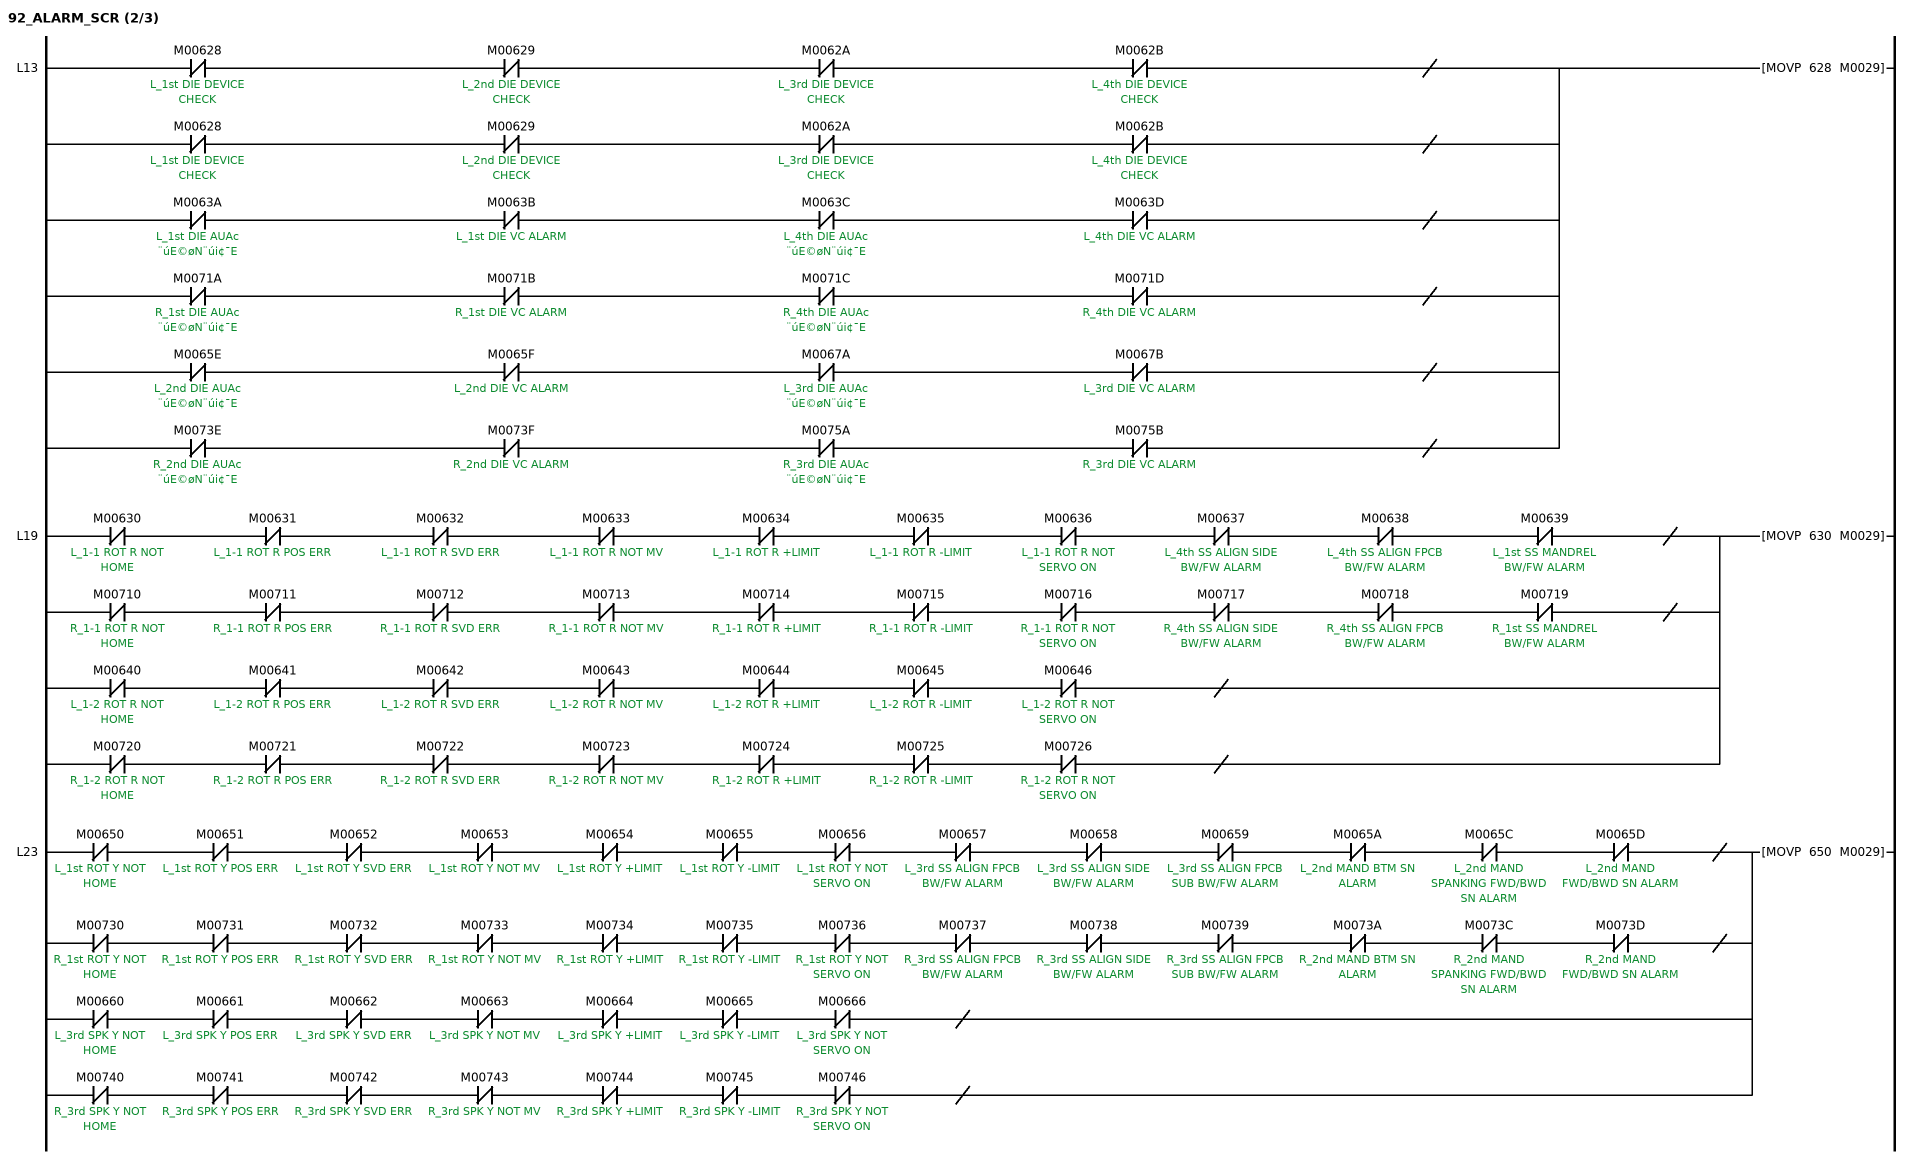
[picture p432: 92_ALARM_SCR rungs L13-L23]
; L13
LOAD NOT  M00628	// L_1st DIE DEVICE CHECK
AND NOT   M00629	// L_2nd DIE DEVICE CHECK
AND NOT   M0062A	// L_3rd DIE DEVICE CHECK
AND NOT   M0062B	// L_4th DIE DEVICE CHECK
NOT
LOAD NOT  M00628	// L_1st DIE DEVICE CHECK
AND NOT   M00629	// L_2nd DIE DEVICE CHECK
AND NOT   M0062A	// L_3rd DIE DEVICE CHECK
AND NOT   M0062B	// L_4th DIE DEVICE CHECK
NOT
OR LOAD
LOAD NOT  M0063A	// L_1st DIE AUAc ¨úE©øN¨úi¢¯E
AND NOT   M0063B	// L_1st DIE VC ALARM
AND NOT   M0063C	// L_4th DIE AUAc ¨úE©øN¨úi¢¯E
AND NOT   M0063D	// L_4th DIE VC ALARM
NOT
OR LOAD
LOAD NOT  M0071A	// R_1st DIE AUAc ¨úE©øN¨úi¢¯E
AND NOT   M0071B	// R_1st DIE VC ALARM
AND NOT   M0071C	// R_4th DIE AUAc ¨úE©øN¨úi¢¯E
AND NOT   M0071D	// R_4th DIE VC ALARM
NOT
OR LOAD
LOAD NOT  M0065E	// L_2nd DIE AUAc ¨úE©øN¨úi¢¯E
AND NOT   M0065F	// L_2nd DIE VC ALARM
AND NOT   M0067A	// L_3rd DIE AUAc ¨úE©øN¨úi¢¯E
AND NOT   M0067B	// L_3rd DIE VC ALARM
NOT
OR LOAD
LOAD NOT  M0073E	// R_2nd DIE AUAc ¨úE©øN¨úi¢¯E
AND NOT   M0073F	// R_2nd DIE VC ALARM
AND NOT   M0075A	// R_3rd DIE AUAc ¨úE©øN¨úi¢¯E
AND NOT   M0075B	// R_3rd DIE VC ALARM
NOT
OR LOAD
MOVP      628 M0029
; L19
LOAD NOT  M00630	// L_1-1 ROT R NOT HOME
AND NOT   M00631	// L_1-1 ROT R POS ERR
AND NOT   M00632	// L_1-1 ROT R SVD ERR
AND NOT   M00633	// L_1-1 ROT R NOT MV
AND NOT   M00634	// L_1-1 ROT R +LIMIT
AND NOT   M00635	// L_1-1 ROT R -LIMIT
AND NOT   M00636	// L_1-1 ROT R NOT SERVO ON
AND NOT   M00637	// L_4th SS ALIGN SIDE BW/FW ALARM
AND NOT   M00638	// L_4th SS ALIGN FPCB BW/FW ALARM
AND NOT   M00639	// L_1st SS MANDREL BW/FW ALARM
NOT
LOAD NOT  M00710	// R_1-1 ROT R NOT HOME
AND NOT   M00711	// R_1-1 ROT R POS ERR
AND NOT   M00712	// R_1-1 ROT R SVD ERR
AND NOT   M00713	// R_1-1 ROT R NOT MV
AND NOT   M00714	// R_1-1 ROT R +LIMIT
AND NOT   M00715	// R_1-1 ROT R -LIMIT
AND NOT   M00716	// R_1-1 ROT R NOT SERVO ON
AND NOT   M00717	// R_4th SS ALIGN SIDE BW/FW ALARM
AND NOT   M00718	// R_4th SS ALIGN FPCB BW/FW ALARM
AND NOT   M00719	// R_1st SS MANDREL BW/FW ALARM
NOT
OR LOAD
LOAD NOT  M00640	// L_1-2 ROT R NOT HOME
AND NOT   M00641	// L_1-2 ROT R POS ERR
AND NOT   M00642	// L_1-2 ROT R SVD ERR
AND NOT   M00643	// L_1-2 ROT R NOT MV
AND NOT   M00644	// L_1-2 ROT R +LIMIT
AND NOT   M00645	// L_1-2 ROT R -LIMIT
AND NOT   M00646	// L_1-2 ROT R NOT SERVO ON
NOT
OR LOAD
LOAD NOT  M00720	// R_1-2 ROT R NOT HOME
AND NOT   M00721	// R_1-2 ROT R POS ERR
AND NOT   M00722	// R_1-2 ROT R SVD ERR
AND NOT   M00723	// R_1-2 ROT R NOT MV
AND NOT   M00724	// R_1-2 ROT R +LIMIT
AND NOT   M00725	// R_1-2 ROT R -LIMIT
AND NOT   M00726	// R_1-2 ROT R NOT SERVO ON
NOT
OR LOAD
MOVP      630 M0029
; L23
LOAD NOT  M00650	// L_1st ROT Y NOT HOME
AND NOT   M00651	// L_1st ROT Y POS ERR
AND NOT   M00652	// L_1st ROT Y SVD ERR
AND NOT   M00653	// L_1st ROT Y NOT MV
AND NOT   M00654	// L_1st ROT Y +LIMIT
AND NOT   M00655	// L_1st ROT Y -LIMIT
AND NOT   M00656	// L_1st ROT Y NOT SERVO ON
AND NOT   M00657	// L_3rd SS ALIGN FPCB BW/FW ALARM
AND NOT   M00658	// L_3rd SS ALIGN SIDE BW/FW ALARM
AND NOT   M00659	// L_3rd SS ALIGN FPCB SUB BW/FW ALARM
AND NOT   M0065A	// L_2nd MAND BTM SN ALARM
AND NOT   M0065C	// L_2nd MAND SPANKING FWD/BWD SN ALARM
AND NOT   M0065D	// L_2nd MAND FWD/BWD SN ALARM
NOT
LOAD NOT  M00730	// R_1st ROT Y NOT HOME
AND NOT   M00731	// R_1st ROT Y POS ERR
AND NOT   M00732	// R_1st ROT Y SVD ERR
AND NOT   M00733	// R_1st ROT Y NOT MV
AND NOT   M00734	// R_1st ROT Y +LIMIT
AND NOT   M00735	// R_1st ROT Y -LIMIT
AND NOT   M00736	// R_1st ROT Y NOT SERVO ON
AND NOT   M00737	// R_3rd SS ALIGN FPCB BW/FW ALARM
AND NOT   M00738	// R_3rd SS ALIGN SIDE BW/FW ALARM
AND NOT   M00739	// R_3rd SS ALIGN FPCB SUB BW/FW ALARM
AND NOT   M0073A	// R_2nd MAND BTM SN ALARM
AND NOT   M0073C	// R_2nd MAND SPANKING FWD/BWD SN ALARM
AND NOT   M0073D	// R_2nd MAND FWD/BWD SN ALARM
NOT
OR LOAD
LOAD NOT  M00660	// L_3rd SPK Y NOT HOME
AND NOT   M00661	// L_3rd SPK Y POS ERR
AND NOT   M00662	// L_3rd SPK Y SVD ERR
AND NOT   M00663	// L_3rd SPK Y NOT MV
AND NOT   M00664	// L_3rd SPK Y +LIMIT
AND NOT   M00665	// L_3rd SPK Y -LIMIT
AND NOT   M00666	// L_3rd SPK Y NOT SERVO ON
NOT
OR LOAD
LOAD NOT  M00740	// R_3rd SPK Y NOT HOME
AND NOT   M00741	// R_3rd SPK Y POS ERR
AND NOT   M00742	// R_3rd SPK Y SVD ERR
AND NOT   M00743	// R_3rd SPK Y NOT MV
AND NOT   M00744	// R_3rd SPK Y +LIMIT
AND NOT   M00745	// R_3rd SPK Y -LIMIT
AND NOT   M00746	// R_3rd SPK Y NOT SERVO ON
NOT
OR LOAD
MOVP      650 M0029

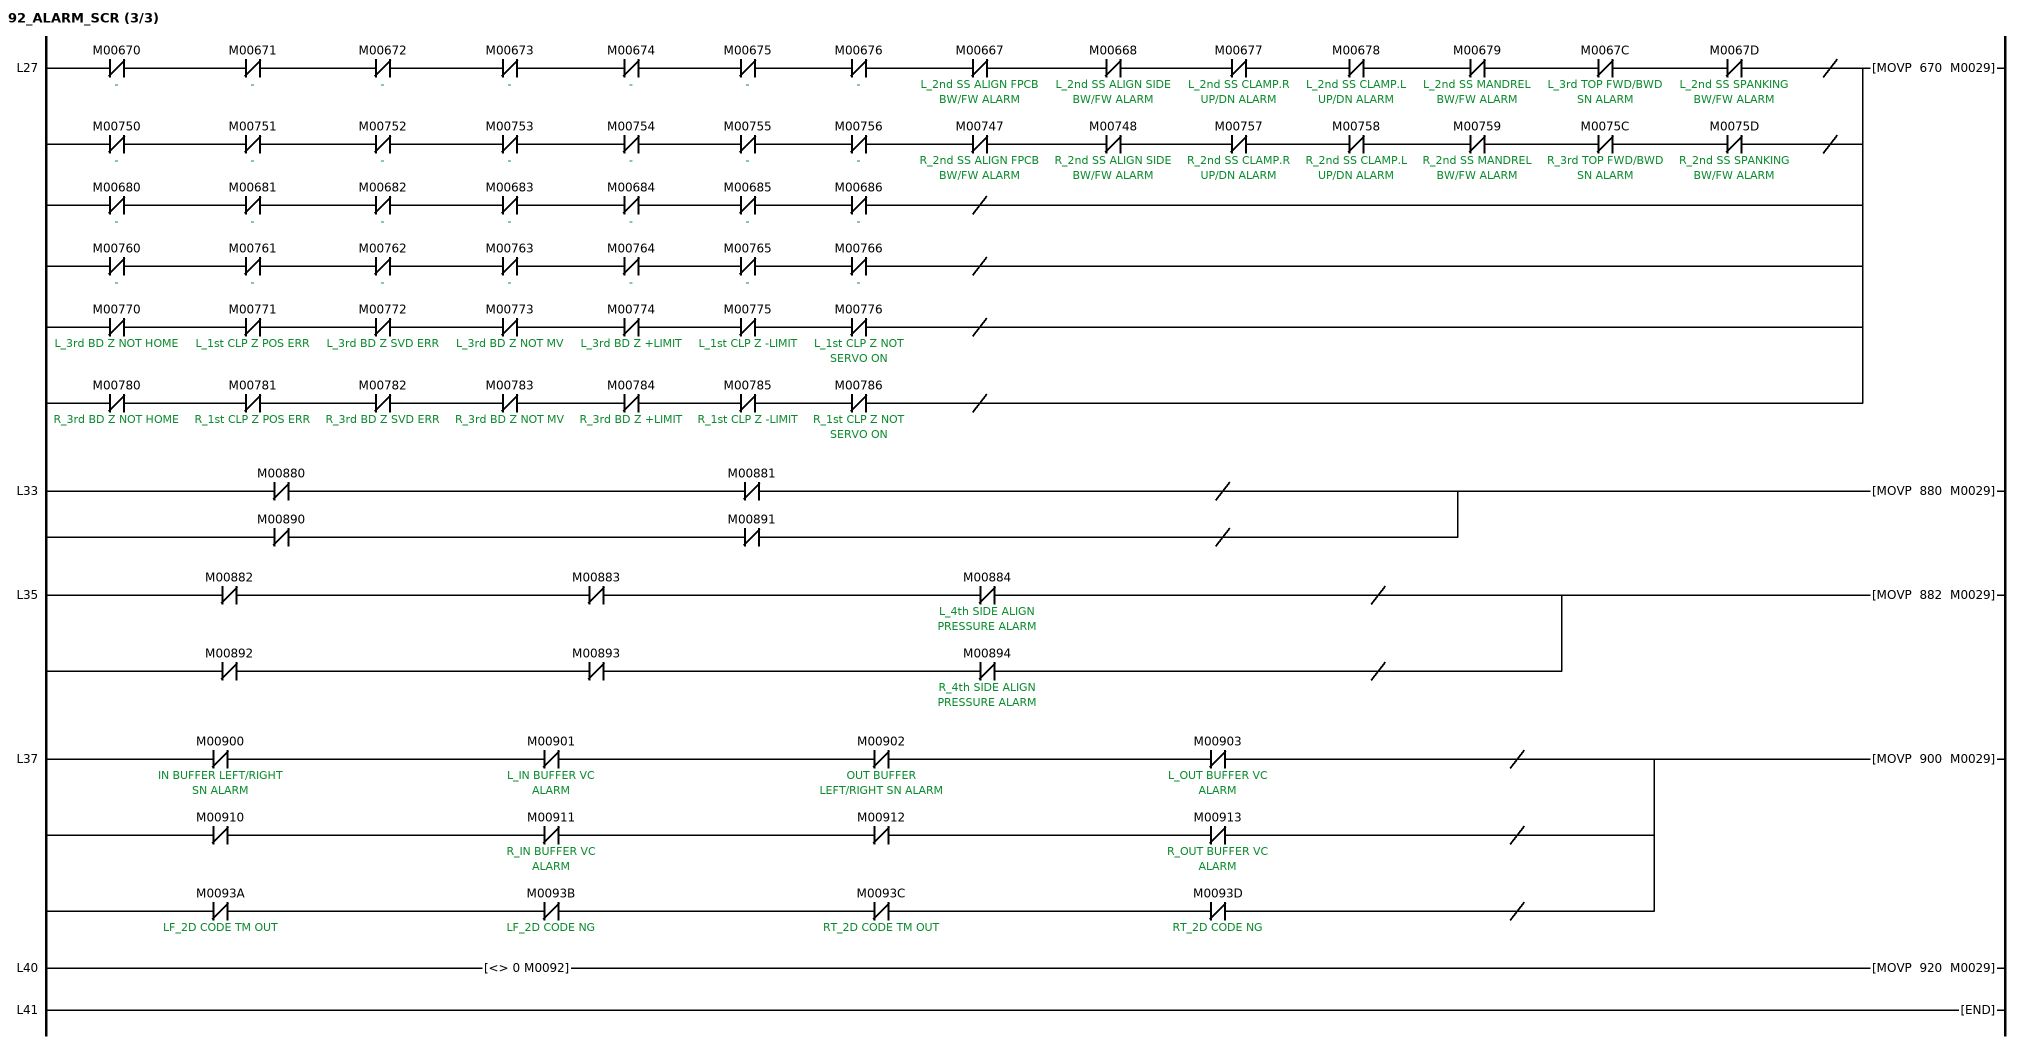
; L27
LOAD NOT  M00670	// -
AND NOT   M00671	// -
AND NOT   M00672	// -
AND NOT   M00673	// -
AND NOT   M00674	// -
AND NOT   M00675	// -
AND NOT   M00676	// -
AND NOT   M00667	// L_2nd SS ALIGN FPCB BW/FW ALARM
AND NOT   M00668	// L_2nd SS ALIGN SIDE BW/FW ALARM
AND NOT   M00677	// L_2nd SS CLAMP.R UP/DN ALARM
AND NOT   M00678	// L_2nd SS CLAMP.L UP/DN ALARM
AND NOT   M00679	// L_2nd SS MANDREL BW/FW ALARM
AND NOT   M0067C	// L_3rd TOP FWD/BWD SN ALARM
AND NOT   M0067D	// L_2nd SS SPANKING BW/FW ALARM
NOT
LOAD NOT  M00750	// -
AND NOT   M00751	// -
AND NOT   M00752	// -
AND NOT   M00753	// -
AND NOT   M00754	// -
AND NOT   M00755	// -
AND NOT   M00756	// -
AND NOT   M00747	// R_2nd SS ALIGN FPCB BW/FW ALARM
AND NOT   M00748	// R_2nd SS ALIGN SIDE BW/FW ALARM
AND NOT   M00757	// R_2nd SS CLAMP.R UP/DN ALARM
AND NOT   M00758	// R_2nd SS CLAMP.L UP/DN ALARM
AND NOT   M00759	// R_2nd SS MANDREL BW/FW ALARM
AND NOT   M0075C	// R_3rd TOP FWD/BWD SN ALARM
AND NOT   M0075D	// R_2nd SS SPANKING BW/FW ALARM
NOT
OR LOAD
LOAD NOT  M00680	// -
AND NOT   M00681	// -
AND NOT   M00682	// -
AND NOT   M00683	// -
AND NOT   M00684	// -
AND NOT   M00685	// -
AND NOT   M00686	// -
NOT
OR LOAD
LOAD NOT  M00760	// -
AND NOT   M00761	// -
AND NOT   M00762	// -
AND NOT   M00763	// -
AND NOT   M00764	// -
AND NOT   M00765	// -
AND NOT   M00766	// -
NOT
OR LOAD
LOAD NOT  M00770	// L_3rd BD Z NOT HOME
AND NOT   M00771	// L_1st CLP Z POS ERR
AND NOT   M00772	// L_3rd BD Z SVD ERR
AND NOT   M00773	// L_3rd BD Z NOT MV
AND NOT   M00774	// L_3rd BD Z +LIMIT
AND NOT   M00775	// L_1st CLP Z -LIMIT
AND NOT   M00776	// L_1st CLP Z NOT SERVO ON
NOT
OR LOAD
LOAD NOT  M00780	// R_3rd BD Z NOT HOME
AND NOT   M00781	// R_1st CLP Z POS ERR
AND NOT   M00782	// R_3rd BD Z SVD ERR
AND NOT   M00783	// R_3rd BD Z NOT MV
AND NOT   M00784	// R_3rd BD Z +LIMIT
AND NOT   M00785	// R_1st CLP Z -LIMIT
AND NOT   M00786	// R_1st CLP Z NOT SERVO ON
NOT
OR LOAD
MOVP      670 M0029
; L33
LOAD NOT  M00880
AND NOT   M00881
NOT
LOAD NOT  M00890
AND NOT   M00891
NOT
OR LOAD
MOVP      880 M0029
; L35
LOAD NOT  M00882
AND NOT   M00883
AND NOT   M00884	// L_4th SIDE ALIGN PRESSURE ALARM
NOT
LOAD NOT  M00892
AND NOT   M00893
AND NOT   M00894	// R_4th SIDE ALIGN PRESSURE ALARM
NOT
OR LOAD
MOVP      882 M0029
; L37
LOAD NOT  M00900	// IN BUFFER LEFT/RIGHT SN ALARM
AND NOT   M00901	// L_IN BUFFER VC ALARM
AND NOT   M00902	// OUT BUFFER LEFT/RIGHT SN ALARM
AND NOT   M00903	// L_OUT BUFFER VC ALARM
NOT
LOAD NOT  M00910
AND NOT   M00911	// R_IN BUFFER VC ALARM
AND NOT   M00912
AND NOT   M00913	// R_OUT BUFFER VC ALARM
NOT
OR LOAD
LOAD NOT  M0093A	// LF_2D CODE TM OUT
AND NOT   M0093B	// LF_2D CODE NG
AND NOT   M0093C	// RT_2D CODE TM OUT
AND NOT   M0093D	// RT_2D CODE NG
NOT
OR LOAD
MOVP      900 M0029
; L40
LOAD<>    0 M0092
MOVP      920 M0029
; L41
END

PROGRAM AUTO_LOAD (task: ¨ö¨¬A¥ì CA¡¤I¡¾¡¿¡¤¡Í)

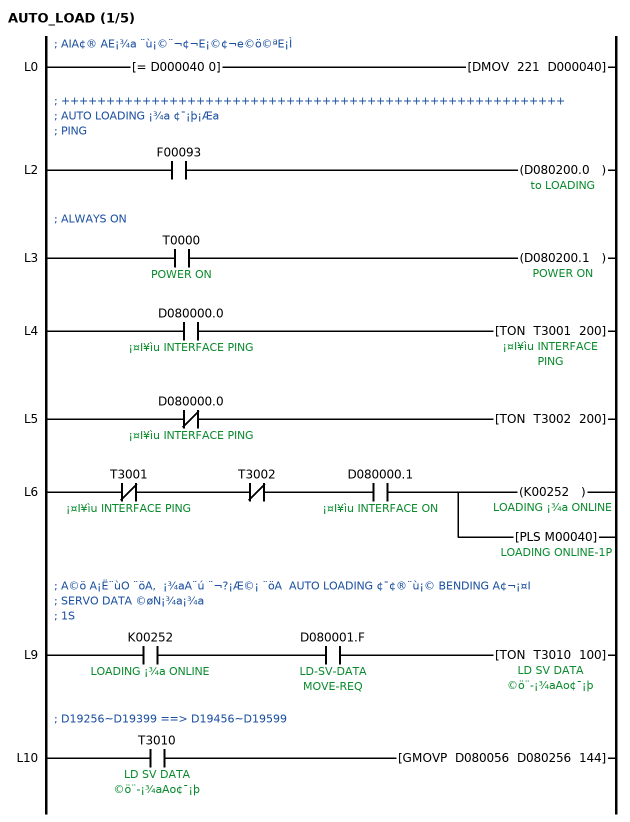
; L0
LOAD=     D000040 0
DMOV      221 D000040
// output comment: AIA¢® AE¡¾a ¨ù¡©¨¬¢¬E¡©¢¬e©ö©ªE¡Ì
// ++++++++++++++++++++++++++++++++++++++++++++++++++++++++
//    AUTO LOADING ¡¾a ¢¯¡þ¡Æa
; L2
LOAD      F00093
OUT       D080200.0	// to LOADING
// output comment: PING
; L3
LOAD      T0000	// POWER ON
OUT       D080200.1	// POWER ON
// output comment: ALWAYS ON
; L4
LOAD      D080000.0	// ¡¤I¥ìu INTERFACE PING
TON       T3001 200	// ¡¤I¥ìu INTERFACE PING
; L5
LOAD NOT  D080000.0	// ¡¤I¥ìu INTERFACE PING
TON       T3002 200
; L6
LOAD NOT  T3001	// ¡¤I¥ìu INTERFACE PING
AND NOT   T3002
AND       D080000.1	// ¡¤I¥ìu INTERFACE ON
OUT       K00252	// LOADING ¡¾a ONLINE
OUTP      M00040	// LOADING ONLINE-1P
// A©ö A¡Ë¨ùO ¨öA,  ¡¾aA¨ú ¨¬?¡Æ©¡ ¨öA  AUTO LOADING ¢¯¢®¨ù¡© BENDING A¢¬¡¤I  SERVO DATA ©øN¡¾a¡¾a
; L9
LOAD      K00252	// LOADING ¡¾a ONLINE
AND       D080001.F	// LD-SV-DATA MOVE-REQ
TON       T3010 100	// LD SV DATA ©ö¨­¡¾aAo¢¯¡þ
// output comment: 1S
; L10
LOAD      T3010	// LD SV DATA ©ö¨­¡¾aAo¢¯¡þ
GMOVP     D080056 D080256 144
// output comment: D19256~D19399 ==> D19456~D19599

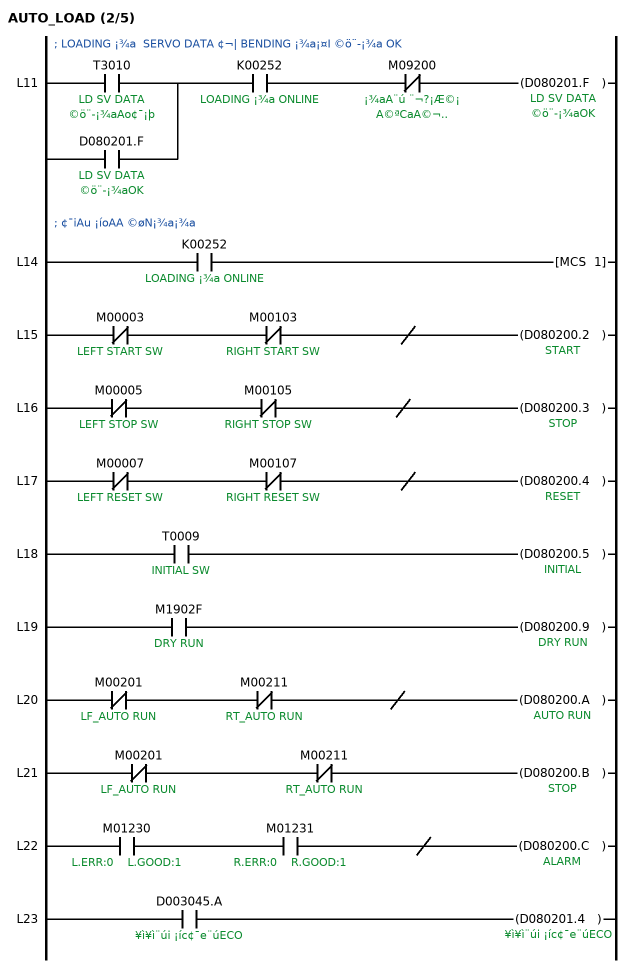
; L11
LOAD      T3010	// LD SV DATA ©ö¨­¡¾aAo¢¯¡þ
OR        D080201.F	// LD SV DATA ©ö¨­¡¾aOK
AND       K00252	// LOADING ¡¾a ONLINE
AND NOT   M09200	// ¡¾aA¨ú ¨¬?¡Æ©¡ A©ªCaA©¬..
OUT       D080201.F	// LD SV DATA ©ö¨­¡¾aOK
// output comment: LOADING ¡¾a  SERVO DATA ¢¬| BENDING ¡¾a¡¤I ©ö¨­¡¾a OK
// ¢¯iAu ¡íoAA ©øN¡¾a¡¾a
; L14
LOAD      K00252	// LOADING ¡¾a ONLINE
MCS       1
; L15
LOAD NOT  M00003	// LEFT START SW
AND NOT   M00103	// RIGHT START SW
NOT
OUT       D080200.2	// START
; L16
LOAD NOT  M00005	// LEFT STOP SW
AND NOT   M00105	// RIGHT STOP SW
NOT
OUT       D080200.3	// STOP
; L17
LOAD NOT  M00007	// LEFT RESET SW
AND NOT   M00107	// RIGHT RESET SW
NOT
OUT       D080200.4	// RESET
; L18
LOAD      T0009	// INITIAL SW
OUT       D080200.5	// INITIAL
; L19
LOAD      M1902F	// DRY RUN
OUT       D080200.9	// DRY RUN
; L20
LOAD NOT  M00201	// LF_AUTO RUN
AND NOT   M00211	// RT_AUTO RUN
NOT
OUT       D080200.A	// AUTO RUN
; L21
LOAD NOT  M00201	// LF_AUTO RUN
AND NOT   M00211	// RT_AUTO RUN
OUT       D080200.B	// STOP
; L22
LOAD      M01230	// L.ERR:0    L.GOOD:1
AND       M01231	// R.ERR:0    R.GOOD:1
NOT
OUT       D080200.C	// ALARM
; L23
LOAD      D003045.A	// ¥ì¥ì¨úi ¡íc¢¯e¨úECO
OUT       D080201.4	// ¥ì¥ì¨úi ¡íc¢¯e¨úECO

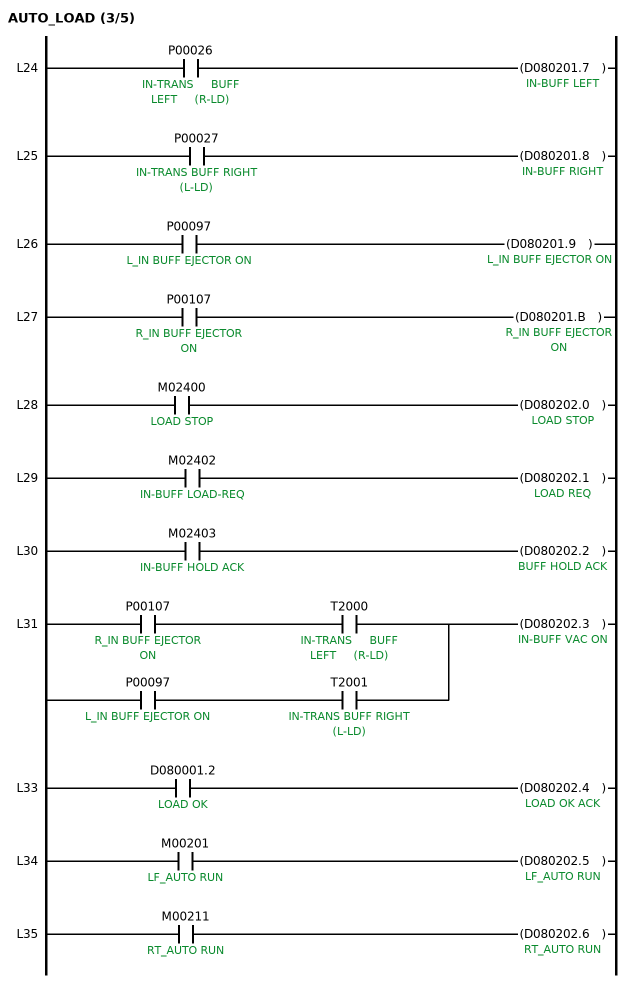
; L24
LOAD      P00026	// IN-TRANS     BUFF     LEFT     (R-LD)
OUT       D080201.7	// IN-BUFF LEFT
; L25
LOAD      P00027	// IN-TRANS BUFF RIGHT     (L-LD)
OUT       D080201.8	// IN-BUFF RIGHT
; L26
LOAD      P00097	// L_IN BUFF EJECTOR ON
OUT       D080201.9	// L_IN BUFF EJECTOR ON
; L27
LOAD      P00107	// R_IN BUFF EJECTOR ON
OUT       D080201.B	// R_IN BUFF EJECTOR ON
; L28
LOAD      M02400	// LOAD STOP
OUT       D080202.0	// LOAD STOP
; L29
LOAD      M02402	// IN-BUFF LOAD-REQ
OUT       D080202.1	// LOAD REQ
; L30
LOAD      M02403	// IN-BUFF HOLD ACK
OUT       D080202.2	// BUFF HOLD ACK
; L31
LOAD      P00107	// R_IN BUFF EJECTOR ON
AND       T2000	// IN-TRANS     BUFF     LEFT     (R-LD)
LOAD      P00097	// L_IN BUFF EJECTOR ON
AND       T2001	// IN-TRANS BUFF RIGHT     (L-LD)
OR LOAD
OUT       D080202.3	// IN-BUFF VAC ON
; L33
LOAD      D080001.2	// LOAD OK
OUT       D080202.4	// LOAD OK ACK
; L34
LOAD      M00201	// LF_AUTO RUN
OUT       D080202.5	// LF_AUTO RUN
; L35
LOAD      M00211	// RT_AUTO RUN
OUT       D080202.6	// RT_AUTO RUN

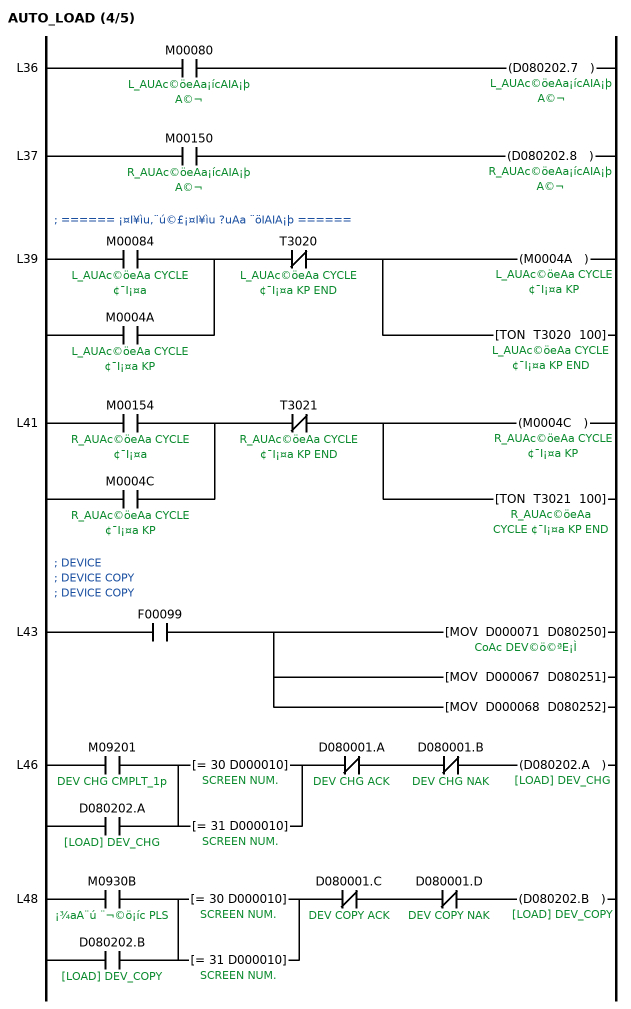
; L36
LOAD      M00080	// L_AUAc©öeAa¡ícAIA¡þA©¬
OUT       D080202.7	// L_AUAc©öeAa¡ícAIA¡þA©¬
; L37
LOAD      M00150	// R_AUAc©öeAa¡ícAIA¡þA©¬
OUT       D080202.8	// R_AUAc©öeAa¡ícAIA¡þA©¬
// ====== ¡¤I¥ìu,¨ú©£¡¤I¥ìu ?uAa ¨öIAIA¡þ ======
; L39
LOAD      M00084	// L_AUAc©öeAa CYCLE ¢¯I¡¤a
OR        M0004A	// L_AUAc©öeAa CYCLE ¢¯I¡¤a KP
AND NOT   T3020	// L_AUAc©öeAa CYCLE ¢¯I¡¤a KP END
OUT       M0004A	// L_AUAc©öeAa CYCLE ¢¯I¡¤a KP
TON       T3020 100	// L_AUAc©öeAa CYCLE ¢¯I¡¤a KP END
; L41
LOAD      M00154	// R_AUAc©öeAa CYCLE ¢¯I¡¤a
OR        M0004C	// R_AUAc©öeAa CYCLE ¢¯I¡¤a KP
AND NOT   T3021	// R_AUAc©öeAa CYCLE ¢¯I¡¤a KP END
OUT       M0004C	// R_AUAc©öeAa CYCLE ¢¯I¡¤a KP
TON       T3021 100	// R_AUAc©öeAa CYCLE ¢¯I¡¤a KP END
; L43
LOAD      F00099
MOV       D000071 D080250	// CoAc DEV©ö©ªE¡Ì
MOV       D000067 D080251
MOV       D000068 D080252
// output comment: DEVICE
// output comment: DEVICE COPY
// output comment: DEVICE COPY
; L46
LOAD      M09201	// DEV CHG CMPLT_1p
OR        D080202.A	// [LOAD] DEV_CHG
LOAD=     30 D000010	// SCREEN NUM.
OR=       31 D000010	// SCREEN NUM.
AND LOAD
AND NOT   D080001.A	// DEV CHG ACK
AND NOT   D080001.B	// DEV CHG NAK
OUT       D080202.A	// [LOAD] DEV_CHG
; L48
LOAD      M0930B	// ¡¾aA¨ú ¨¬©ö¡íc PLS
OR        D080202.B	// [LOAD] DEV_COPY
LOAD=     30 D000010	// SCREEN NUM.
OR=       31 D000010	// SCREEN NUM.
AND LOAD
AND NOT   D080001.C	// DEV COPY ACK
AND NOT   D080001.D	// DEV COPY NAK
OUT       D080202.B	// [LOAD] DEV_COPY

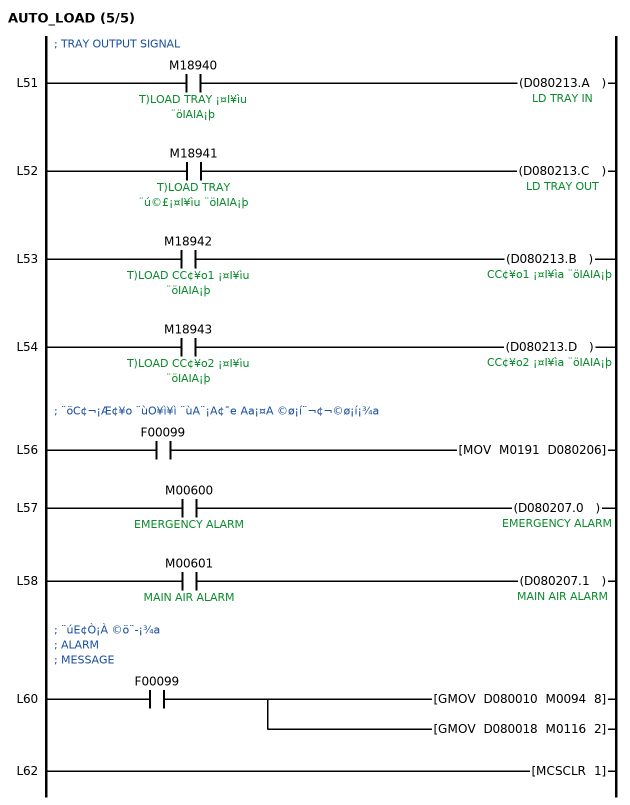
// TRAY OUTPUT SIGNAL
; L51
LOAD      M18940	// T)LOAD TRAY ¡¤I¥ìu ¨öIAIA¡þ
OUT       D080213.A	// LD TRAY IN
; L52
LOAD      M18941	// T)LOAD TRAY ¨ú©£¡¤I¥ìu ¨öIAIA¡þ
OUT       D080213.C	// LD TRAY OUT
; L53
LOAD      M18942	// T)LOAD CC¢¥o1 ¡¤I¥ìu ¨öIAIA¡þ
OUT       D080213.B	// CC¢¥o1 ¡¤I¥ìa ¨öIAIA¡þ
; L54
LOAD      M18943	// T)LOAD CC¢¥o2 ¡¤I¥ìu ¨öIAIA¡þ
OUT       D080213.D	// CC¢¥o2 ¡¤I¥ìa ¨öIAIA¡þ
// ¨öC¢¬¡Æ¢¥o ¨ùO¥ì¥ì ¨ùA¨¡A¢¯e Aa¡¤A ©ø¡í¨¬¢¬©ø¡í¡¾a
; L56
LOAD      F00099
MOV       M0191 D080206
; L57
LOAD      M00600	// EMERGENCY ALARM
OUT       D080207.0	// EMERGENCY ALARM
; L58
LOAD      M00601	// MAIN AIR ALARM
OUT       D080207.1	// MAIN AIR ALARM
// ¨úE¢Ò¡À ©ö¨­¡¾a
; L60
LOAD      F00099
GMOV      D080010 M0094 8
GMOV      D080018 M0116 2
// output comment: ALARM
// output comment: MESSAGE
; L62
MCSCLR    1

PROGRAM AUTO_UNLOAD (task: ¨ö¨¬A¥ì CA¡¤I¡¾¡¿¡¤¡Í)

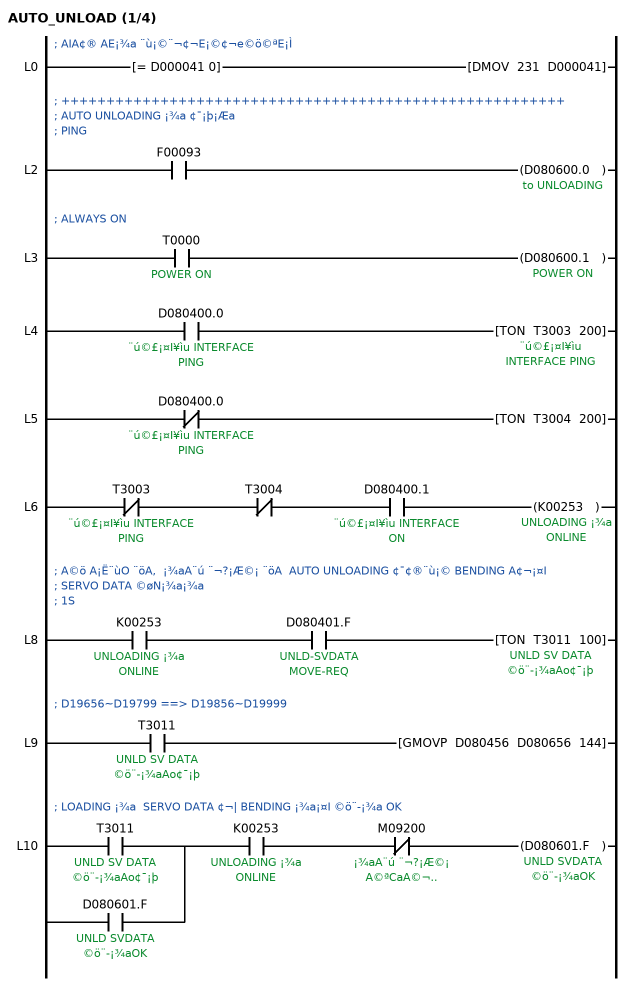
; L0
LOAD=     D000041 0
DMOV      231 D000041
// output comment: AIA¢® AE¡¾a ¨ù¡©¨¬¢¬E¡©¢¬e©ö©ªE¡Ì
// ++++++++++++++++++++++++++++++++++++++++++++++++++++++++
//    AUTO UNLOADING ¡¾a ¢¯¡þ¡Æa
; L2
LOAD      F00093
OUT       D080600.0	// to UNLOADING
// output comment: PING
; L3
LOAD      T0000	// POWER ON
OUT       D080600.1	// POWER ON
// output comment: ALWAYS ON
; L4
LOAD      D080400.0	// ¨ú©£¡¤I¥ìu INTERFACE PING
TON       T3003 200	// ¨ú©£¡¤I¥ìu INTERFACE PING
; L5
LOAD NOT  D080400.0	// ¨ú©£¡¤I¥ìu INTERFACE PING
TON       T3004 200
; L6
LOAD NOT  T3003	// ¨ú©£¡¤I¥ìu INTERFACE PING
AND NOT   T3004
AND       D080400.1	// ¨ú©£¡¤I¥ìu INTERFACE ON
OUT       K00253	// UNLOADING ¡¾a ONLINE
// A©ö A¡Ë¨ùO ¨öA,  ¡¾aA¨ú ¨¬?¡Æ©¡ ¨öA  AUTO UNLOADING ¢¯¢®¨ù¡© BENDING A¢¬¡¤I  SERVO DATA ©øN¡¾a¡¾a
; L8
LOAD      K00253	// UNLOADING ¡¾a ONLINE
AND       D080401.F	// UNLD-SVDATA MOVE-REQ
TON       T3011 100	// UNLD SV DATA ©ö¨­¡¾aAo¢¯¡þ
// output comment: 1S
; L9
LOAD      T3011	// UNLD SV DATA ©ö¨­¡¾aAo¢¯¡þ
GMOVP     D080456 D080656 144
// output comment: D19656~D19799 ==> D19856~D19999
; L10
LOAD      T3011	// UNLD SV DATA ©ö¨­¡¾aAo¢¯¡þ
OR        D080601.F	// UNLD SVDATA ©ö¨­¡¾aOK
AND       K00253	// UNLOADING ¡¾a ONLINE
AND NOT   M09200	// ¡¾aA¨ú ¨¬?¡Æ©¡ A©ªCaA©¬..
OUT       D080601.F	// UNLD SVDATA ©ö¨­¡¾aOK
// output comment: LOADING ¡¾a  SERVO DATA ¢¬| BENDING ¡¾a¡¤I ©ö¨­¡¾a OK

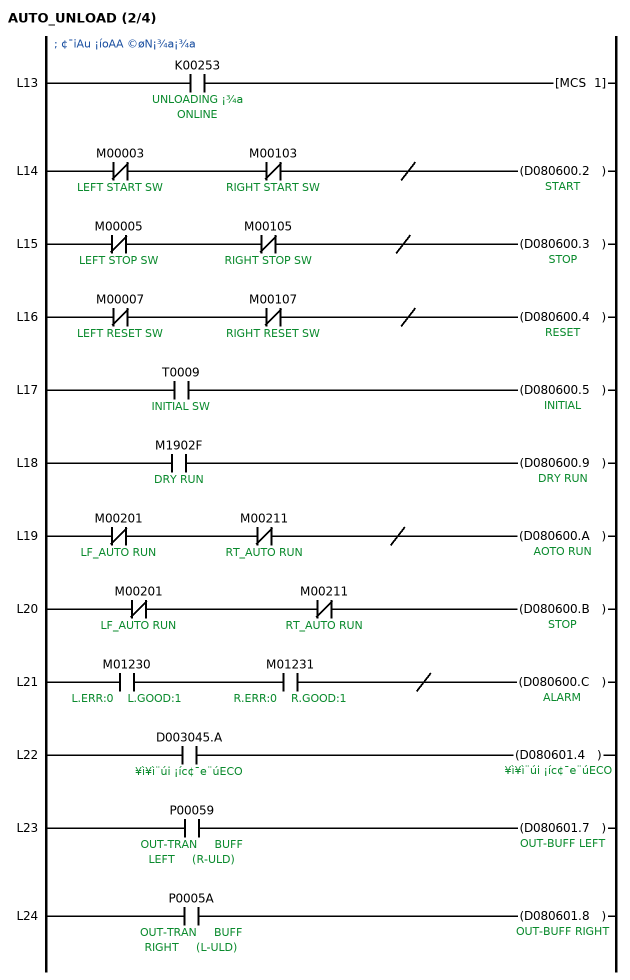
// ¢¯iAu ¡íoAA ©øN¡¾a¡¾a
; L13
LOAD      K00253	// UNLOADING ¡¾a ONLINE
MCS       1
; L14
LOAD NOT  M00003	// LEFT START SW
AND NOT   M00103	// RIGHT START SW
NOT
OUT       D080600.2	// START
; L15
LOAD NOT  M00005	// LEFT STOP SW
AND NOT   M00105	// RIGHT STOP SW
NOT
OUT       D080600.3	// STOP
; L16
LOAD NOT  M00007	// LEFT RESET SW
AND NOT   M00107	// RIGHT RESET SW
NOT
OUT       D080600.4	// RESET
; L17
LOAD      T0009	// INITIAL SW
OUT       D080600.5	// INITIAL
; L18
LOAD      M1902F	// DRY RUN
OUT       D080600.9	// DRY RUN
; L19
LOAD NOT  M00201	// LF_AUTO RUN
AND NOT   M00211	// RT_AUTO RUN
NOT
OUT       D080600.A	// AOTO RUN
; L20
LOAD NOT  M00201	// LF_AUTO RUN
AND NOT   M00211	// RT_AUTO RUN
OUT       D080600.B	// STOP
; L21
LOAD      M01230	// L.ERR:0    L.GOOD:1
AND       M01231	// R.ERR:0    R.GOOD:1
NOT
OUT       D080600.C	// ALARM
; L22
LOAD      D003045.A	// ¥ì¥ì¨úi ¡íc¢¯e¨úECO
OUT       D080601.4	// ¥ì¥ì¨úi ¡íc¢¯e¨úECO
; L23
LOAD      P00059	// OUT-TRAN     BUFF     LEFT     (R-ULD)
OUT       D080601.7	// OUT-BUFF LEFT
; L24
LOAD      P0005A	// OUT-TRAN     BUFF     RIGHT     (L-ULD)
OUT       D080601.8	// OUT-BUFF RIGHT

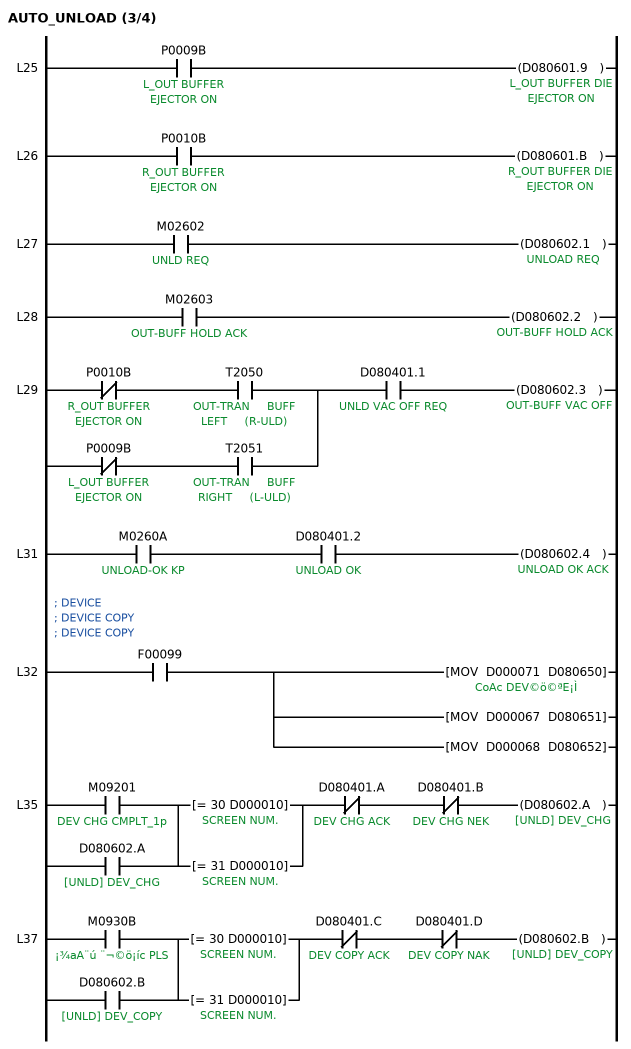
; L25
LOAD      P0009B	// L_OUT BUFFER EJECTOR ON
OUT       D080601.9	// L_OUT BUFFER DIE EJECTOR ON
; L26
LOAD      P0010B	// R_OUT BUFFER EJECTOR ON
OUT       D080601.B	// R_OUT BUFFER DIE EJECTOR ON
; L27
LOAD      M02602	// UNLD REQ
OUT       D080602.1	// UNLOAD REQ
; L28
LOAD      M02603	// OUT-BUFF HOLD ACK
OUT       D080602.2	// OUT-BUFF HOLD ACK
; L29
LOAD NOT  P0010B	// R_OUT BUFFER EJECTOR ON
AND       T2050	// OUT-TRAN     BUFF     LEFT     (R-ULD)
LOAD NOT  P0009B	// L_OUT BUFFER EJECTOR ON
AND       T2051	// OUT-TRAN     BUFF     RIGHT     (L-ULD)
OR LOAD
AND       D080401.1	// UNLD VAC OFF REQ
OUT       D080602.3	// OUT-BUFF VAC OFF
; L31
LOAD      M0260A	// UNLOAD-OK KP
AND       D080401.2	// UNLOAD OK
OUT       D080602.4	// UNLOAD OK ACK
; L32
LOAD      F00099
MOV       D000071 D080650	// CoAc DEV©ö©ªE¡Ì
MOV       D000067 D080651
MOV       D000068 D080652
// output comment: DEVICE
// output comment: DEVICE COPY
// output comment: DEVICE COPY
; L35
LOAD      M09201	// DEV CHG CMPLT_1p
OR        D080602.A	// [UNLD] DEV_CHG
LOAD=     30 D000010	// SCREEN NUM.
OR=       31 D000010	// SCREEN NUM.
AND LOAD
AND NOT   D080401.A	// DEV CHG ACK
AND NOT   D080401.B	// DEV CHG NEK
OUT       D080602.A	// [UNLD] DEV_CHG
; L37
LOAD      M0930B	// ¡¾aA¨ú ¨¬©ö¡íc PLS
OR        D080602.B	// [UNLD] DEV_COPY
LOAD=     30 D000010	// SCREEN NUM.
OR=       31 D000010	// SCREEN NUM.
AND LOAD
AND NOT   D080401.C	// DEV COPY ACK
AND NOT   D080401.D	// DEV COPY NAK
OUT       D080602.B	// [UNLD] DEV_COPY

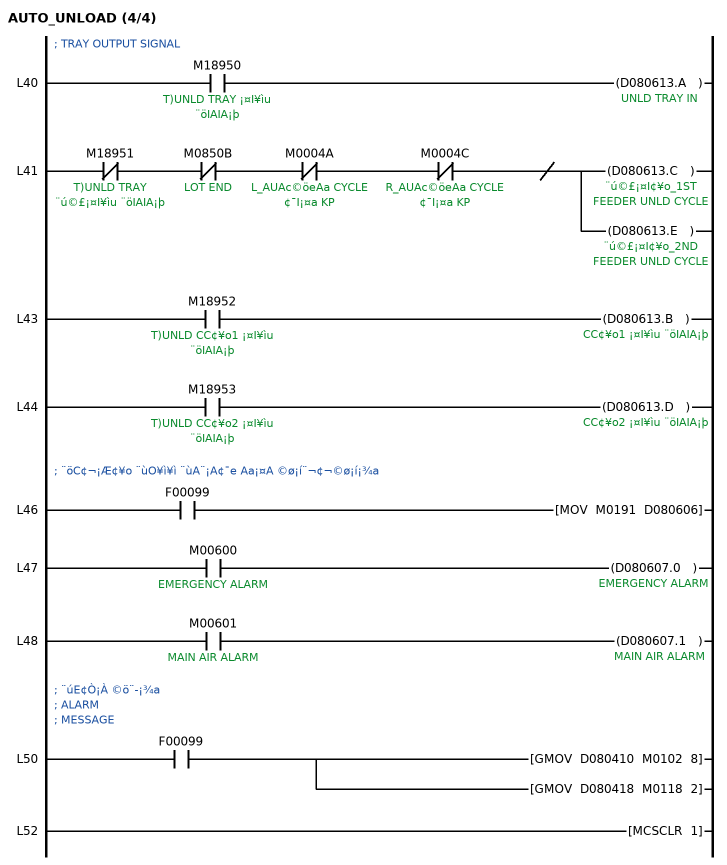
// TRAY OUTPUT SIGNAL
; L40
LOAD      M18950	// T)UNLD TRAY ¡¤I¥ìu ¨öIAIA¡þ
OUT       D080613.A	// UNLD TRAY IN
; L41
LOAD NOT  M18951	// T)UNLD TRAY ¨ú©£¡¤I¥ìu ¨öIAIA¡þ
AND NOT   M0850B	// LOT END 
AND NOT   M0004A	// L_AUAc©öeAa CYCLE ¢¯I¡¤a KP
AND NOT   M0004C	// R_AUAc©öeAa CYCLE ¢¯I¡¤a KP
NOT
OUT       D080613.C	// ¨ú©£¡¤I¢¥o_1ST FEEDER UNLD CYCLE
OUT       D080613.E	// ¨ú©£¡¤I¢¥o_2ND FEEDER UNLD CYCLE
; L43
LOAD      M18952	// T)UNLD CC¢¥o1 ¡¤I¥ìu ¨öIAIA¡þ
OUT       D080613.B	// CC¢¥o1 ¡¤I¥ìu ¨öIAIA¡þ
; L44
LOAD      M18953	// T)UNLD CC¢¥o2 ¡¤I¥ìu ¨öIAIA¡þ
OUT       D080613.D	// CC¢¥o2 ¡¤I¥ìu ¨öIAIA¡þ
// ¨öC¢¬¡Æ¢¥o ¨ùO¥ì¥ì ¨ùA¨¡A¢¯e Aa¡¤A ©ø¡í¨¬¢¬©ø¡í¡¾a
; L46
LOAD      F00099
MOV       M0191 D080606
; L47
LOAD      M00600	// EMERGENCY ALARM
OUT       D080607.0	// EMERGENCY ALARM
; L48
LOAD      M00601	// MAIN AIR ALARM
OUT       D080607.1	// MAIN AIR ALARM
// ¨úE¢Ò¡À ©ö¨­¡¾a
; L50
LOAD      F00099
GMOV      D080410 M0102 8
GMOV      D080418 M0118 2
// output comment: ALARM
// output comment: MESSAGE
; L52
MCSCLR    1

VARIABLES AND COMMENTS (devices not used above)
M10050	BIT	-
M10051	BIT	-
M10052	BIT	-
M10053	BIT	-
M10054	BIT	-
M10055	BIT	-
M10056	BIT	-
M10057	BIT	-
M10058	BIT	-
M10059	BIT	-
M1005A	BIT	-
M1005B	BIT	-
M1005C	BIT	-
M1005D	BIT	-
M1005E	BIT	-
M1005F	BIT	-
M10068	BIT	-
M10069	BIT	-
M1006A	BIT	-
M1006B	BIT	-
M1006C	BIT	-
M1006D	BIT	-
M1006E	BIT	-
M1006F	BIT	-
M10077	BIT	L_1st MAND STEP INITIAL LAMP
M1008C	BIT	L_1st MAND MANUAL SERCH PLS
M1009C	BIT	L_1st MAND ORIGIN ->
M10550	BIT	-
M10551	BIT	-
M10552	BIT	-
M10553	BIT	-
M10554	BIT	-
M10555	BIT	-
M10556	BIT	-
M10557	BIT	-
M10558	BIT	-
M10559	BIT	-
M1055A	BIT	-
M1055B	BIT	-
M1055C	BIT	-
M1055D	BIT	-
M1055E	BIT	-
M1055F	BIT	-
M1056A	BIT	-
M1056B	BIT	-
M1056C	BIT	-
M1056D	BIT	-
M1056E	BIT	-
M1056F	BIT	-
M10577	BIT	L_2nd MAND STEP INITIAL LAMP
M1058C	BIT	L_2nd MAND MANUAL SERCH PLS
M1059C	BIT	L_2nd MAND ORIGIN ->
M1059D	BIT	L_2nd MAND ORIGIN MV ->
M11050	BIT	-
M11051	BIT	-
M11052	BIT	-
M11053	BIT	-
M11054	BIT	-
M11055	BIT	-
M11056	BIT	-
M11057	BIT	-
M11058	BIT	-
M11059	BIT	-
M1105A	BIT	-
M1105B	BIT	-
M1105C	BIT	-
M1105D	BIT	-
M1105E	BIT	-
M1105F	BIT	-
M11068	BIT	-
M11069	BIT	-
M1106A	BIT	-
M1106B	BIT	-
M1106C	BIT	-
M1106D	BIT	-
M1106E	BIT	-
M1106F	BIT	-
M11077	BIT	L_3rd MAND STEP INITIAL LAMP
M1108C	BIT	L_3rd MAND MANUAL SERCH PLS
M1109C	BIT	L_3rd MAND ORIGIN ->
M11550	BIT	-
M11551	BIT	-
M11552	BIT	-
M11553	BIT	-
M11554	BIT	-
M11555	BIT	-
M11556	BIT	-
M11557	BIT	-
M11558	BIT	-
M11559	BIT	-
M1155A	BIT	-
M1155B	BIT	-
M1155C	BIT	-
M1155D	BIT	-
M1155E	BIT	-
M1155F	BIT	-
M11565	BIT	-
M11566	BIT	-
M11567	BIT	-
M11568	BIT	-
M11569	BIT	-
M1156A	BIT	-
M1156B	BIT	-
M1156C	BIT	-
M1156D	BIT	-
M1156E	BIT	-
M1156F	BIT	-
M11577	BIT	L_TOOL STEP INITIAL LAMP
M1158C	BIT	L_TOOL MANUAL SERCH PLS
M1159C	BIT	L_TOOL ORIGIN ->
M1159D	BIT	L_TOOL ORIGIN MV ->
M12020	BIT	L_P&P STEP#16
M12021	BIT	L_P&P STEP#17
M12022	BIT	L_P&P STEP#18
M12023	BIT	L_P&P STEP#19
M12024	BIT	L_P&P STEP#20
M12025	BIT	L_P&P STEP#21
M12026	BIT	L_P&P STEP#22
M12027	BIT	L_P&P STEP#23
M12028	BIT	L_P&P STEP#24
M12029	BIT	L_P&P STEP#25
M1202A	BIT	L_P&P STEP#26
M1202B	BIT	L_P&P STEP#27
M1202C	BIT	L_P&P STEP#28
M1202D	BIT	L_P&P STEP#29
M1202E	BIT	L_P&P STEP#30
M1202F	BIT	L_P&P STEP#31
M12040	BIT	STEP A¢Ò¡ÆC16
M12041	BIT	STEP A¢Ò¡ÆC17
M12042	BIT	STEP A¢Ò¡ÆC18
M12043	BIT	STEP A¢Ò¡ÆC19
M12044	BIT	STEP A¢Ò¡ÆC20
M12045	BIT	STEP A¢Ò¡ÆC21
M12046	BIT	STEP A¢Ò¡ÆC22
M12047	BIT	STEP A¢Ò¡ÆC23
M12048	BIT	STEP A¢Ò¡ÆC24
M12049	BIT	STEP A¢Ò¡ÆC25
M1204A	BIT	STEP A¢Ò¡ÆC26
M1204B	BIT	STEP A¢Ò¡ÆC27
M1204C	BIT	STEP A¢Ò¡ÆC28
M1204D	BIT	STEP A¢Ò¡ÆC29
M1204E	BIT	STEP A¢Ò¡ÆC30
M1204F	BIT	STEP A¢Ò¡ÆC31
M12050	BIT	-
M12051	BIT	-
M12052	BIT	-
M12053	BIT	-
M12054	BIT	-
M12055	BIT	-
M12056	BIT	-
M12057	BIT	-
M12058	BIT	-
M12059	BIT	-
M1205A	BIT	-
M1205B	BIT	-
M1205C	BIT	-
M1205D	BIT	-
M1205E	BIT	-
M1205F	BIT	-
M12062	BIT	-
M12063	BIT	-
M12064	BIT	-
M12065	BIT	-
M12066	BIT	-
M12067	BIT	-
M12068	BIT	-
M12069	BIT	-
M1206A	BIT	-
M1206B	BIT	-
M1206C	BIT	-
M1206D	BIT	-
M1206E	BIT	-
M1206F	BIT	-
M12077	BIT	L_P&P STEP INITIAL LAMP
M1208C	BIT	L_P&P MANUAL SERCH PLS
M1209C	BIT	L_P&P ORIGIN ->
M12550	BIT	-
M12551	BIT	-
M12552	BIT	-
M12553	BIT	-
M12554	BIT	-
M12555	BIT	-
M12556	BIT	-
M12557	BIT	-
M12558	BIT	-
M12559	BIT	-
M1255A	BIT	-
M1255B	BIT	-
M1255C	BIT	-
M1255D	BIT	-
M1255E	BIT	-
M1255F	BIT	-
M12568	BIT	-
M12569	BIT	-
M1256A	BIT	-
M1256B	BIT	-
M1256C	BIT	-
M1256D	BIT	-
M1256E	BIT	-
M1256F	BIT	-
M12577	BIT	R_1st MAND STEP INITIAL LAMP
M1258C	BIT	R_1st MAND MANUAL SERCH PLS
M1259C	BIT	R_1st MAND ORIGIN ->
M1259D	BIT	R_1st MAND ORIGIN MV ->
M13050	BIT	-
M13051	BIT	-
M13052	BIT	-
M13053	BIT	-
M13054	BIT	-
M13055	BIT	-
M13056	BIT	-
M13057	BIT	-
M13058	BIT	-
M13059	BIT	-
M1305A	BIT	-
M1305B	BIT	-
M1305C	BIT	-
M1305D	BIT	-
M1305E	BIT	-
M1305F	BIT	-
M1306A	BIT	-
M1306B	BIT	-
M1306C	BIT	-
M1306D	BIT	-
M1306E	BIT	-
M1306F	BIT	-
M13077	BIT	R_2nd MAND STEP INITIAL LAMP
M1308C	BIT	R_2nd MAND MANUAL SERCH PLS
M1309C	BIT	R_2nd MAND ORIGIN ->
M13550	BIT	-
M13551	BIT	-
M13552	BIT	-
M13553	BIT	-
M13554	BIT	-
M13555	BIT	-
M13556	BIT	-
M13557	BIT	-
M13558	BIT	-
M13559	BIT	-
M1355A	BIT	-
M1355B	BIT	-
M1355C	BIT	-
M1355D	BIT	-
M1355E	BIT	-
M1355F	BIT	-
M13568	BIT	-
M13569	BIT	-
M1356A	BIT	-
M1356B	BIT	-
M1356C	BIT	-
M1356D	BIT	-
M1356E	BIT	-
M1356F	BIT	-
M13577	BIT	R_3rd MAND STEP INITIAL LAMP
M1358C	BIT	R_3rd MAND MANUAL SERCH PLS
M1359C	BIT	R_3rd MAND ORIGIN ->
M14050	BIT	-
M14051	BIT	-
M14052	BIT	-
M14053	BIT	-
M14054	BIT	-
M14055	BIT	-
M14056	BIT	-
M14057	BIT	-
M14058	BIT	-
M14059	BIT	-
M1405A	BIT	-
M1405B	BIT	-
M1405C	BIT	-
M1405D	BIT	-
M1405E	BIT	-
M1405F	BIT	-
M14066	BIT	-
M14067	BIT	-
M14068	BIT	-
M14069	BIT	-
M1406A	BIT	-
M1406B	BIT	-
M1406C	BIT	-
M1406D	BIT	-
M1406E	BIT	-
M1406F	BIT	-
M14077	BIT	R_TOOL STEP INITIAL LAMP
M1408C	BIT	R_TOOL MANUAL SERCH PLS
M1409C	BIT	R_TOOL ORIGIN ->
M14520	BIT	R_P&P STEP#16
M14521	BIT	R_P&P STEP#17
M14522	BIT	R_P&P STEP#18
M14523	BIT	R_P&P STEP#19
M14524	BIT	R_P&P STEP#20
M14525	BIT	R_P&P STEP#21
M14526	BIT	R_P&P STEP#22
M14527	BIT	R_P&P STEP#23
M14528	BIT	R_P&P STEP#24
M14529	BIT	R_P&P STEP#25
M1452A	BIT	R_P&P STEP#26
M1452B	BIT	R_P&P STEP#27
M1452C	BIT	R_P&P STEP#28
M1452D	BIT	R_P&P STEP#29
M1452E	BIT	R_P&P STEP#30
M1452F	BIT	R_P&P STEP#31
M14540	BIT	STEP A¢Ò¡ÆC16
M14541	BIT	STEP A¢Ò¡ÆC17
M14542	BIT	STEP A¢Ò¡ÆC18
M14543	BIT	STEP A¢Ò¡ÆC19
M14544	BIT	STEP A¢Ò¡ÆC20
M14545	BIT	STEP A¢Ò¡ÆC21
M14546	BIT	STEP A¢Ò¡ÆC22
M14547	BIT	STEP A¢Ò¡ÆC23
M14548	BIT	STEP A¢Ò¡ÆC24
M14549	BIT	STEP A¢Ò¡ÆC25
M1454A	BIT	STEP A¢Ò¡ÆC26
M1454B	BIT	STEP A¢Ò¡ÆC27
M1454C	BIT	STEP A¢Ò¡ÆC28
M1454D	BIT	STEP A¢Ò¡ÆC29
M1454E	BIT	STEP A¢Ò¡ÆC30
M1454F	BIT	STEP A¢Ò¡ÆC31
M14550	BIT	-
M14551	BIT	-
M14552	BIT	-
M14553	BIT	-
M14554	BIT	-
M14555	BIT	-
M14556	BIT	-
M14557	BIT	-
M14558	BIT	-
M14559	BIT	-
M1455A	BIT	-
M1455B	BIT	-
M1455C	BIT	-
M1455D	BIT	-
M1455E	BIT	-
M1455F	BIT	-
M14562	BIT	-
M14563	BIT	-
M14564	BIT	-
M14565	BIT	-
M14566	BIT	-
M14567	BIT	-
M14568	BIT	-
M14569	BIT	-
M1456A	BIT	-
M1456B	BIT	-
M1456C	BIT	-
M1456D	BIT	-
M1456E	BIT	-
M1456F	BIT	-
M14577	BIT	R_P&P STEP INITIAL LAMP
M1458C	BIT	R_P&P MANUAL SERCH PLS
M1459C	BIT	R_P&P ORIGIN ->
M01516	BIT	L_4th BD Z SPD MV PLS
M01517	BIT	L_4th BD Z SPD OVERRIDE PLS
M01518	BIT	L_4th BD Z HOME ENABLE
M01519	BIT	L_4th BD Z HOME ->
M0151B	BIT	L_4th BD Z SPD START
M01526	BIT	L_P&P Y SPD MV PLS
M01527	BIT	L_P&P Y SPD OVERRIDE PLS
M01528	BIT	L_P&P Y HOME ENABLE
M01529	BIT	L_P&P Y HOME ->
M0152B	BIT	L_P&P Y SPD START
M01536	BIT	L_1-1 ROT R SPD MV PLS
M01537	BIT	L_1-1 ROT R SPD OVERRIDE PLS
M01538	BIT	L_1-1 ROT R HOME ENABLE
M01539	BIT	L_1-1 ROT R HOME ->
M0153B	BIT	L_1-1 ROT R SPD START
M01546	BIT	L_1-2 ROT R SPD MV PLS
M01547	BIT	L_1-2 ROT R OVERRIDE PLS
M01548	BIT	L_1-2 ROT R HOME ENABLE
M01549	BIT	L_1-2 ROT R HOME ->
M0154B	BIT	L_1-2 ROT R START
M01556	BIT	L_1st ROT Y SPD MV PLS
M01557	BIT	L_1st ROT Y OVERRIDE PLS
M01558	BIT	L_1st ROT Y HOME ENABLE
M01559	BIT	L_1st ROT Y HOME ->
M0155B	BIT	L_1st ROT Y START
M01566	BIT	L_3rd SPK Y SPD MV PLS
M01567	BIT	L_3rd SPK Y OVERRIDE PLS
M01568	BIT	L_3rd SPK Y HOME ENABLE
M01569	BIT	L_3rd SPK Y HOME ->
M0156B	BIT	L_3rd SPK Y START
M01576	BIT	-
M01577	BIT	-
M01578	BIT	-
M01579	BIT	-
M0157B	BIT	-
M01586	BIT	-
M01587	BIT	-
M01588	BIT	-
M01589	BIT	-
M0158B	BIT	-
M01596	BIT	R_4th BD Z SPD MV PLS
M01597	BIT	R_4th BD Z OVERRIDE PLS
M01598	BIT	R_4th BD Z HOME ENABLE
M01599	BIT	R_4th BD Z HOME ->
M0159B	BIT	R_4th BD Z START
M01606	BIT	R_P&P Y SPD MV PLS
M01607	BIT	R_P&P Y OVERRIDE PLS
M01608	BIT	R_P&P Y HOME ENABLE
M01609	BIT	R_P&P Y HOME ->
M0160B	BIT	R_P&P Y START
M01616	BIT	R_1-1 ROT R SPD MV PLS
M01617	BIT	R_1-1 ROT R OVERRIDE PLS
M01618	BIT	R_1-1 ROT R HOME ENABLE
M01619	BIT	R_1-1 ROT R HOME ->
M0161B	BIT	R_1-1 ROT R START
M01626	BIT	R_1-2 ROT R SPD MV PLS
M01627	BIT	R_1-2 ROT R OVERRIDE PLS
M01628	BIT	R_1-2 ROT R HOME ENABLE
M01629	BIT	R_1-2 ROT R HOME ->
M0162B	BIT	R_1-2 ROT R START
M01636	BIT	R_1st ROT Y SPD MV PLS
M01637	BIT	R_1st ROT Y OVERRIDE PLS
M01638	BIT	R_1st ROT Y HOME ENABLE
M01639	BIT	R_1st ROT Y HOME ->
M0163B	BIT	R_1st ROT Y START
M01646	BIT	R_3rd SPK Y SPD MV PLS
M01647	BIT	R_3rd SPK Y OVERRIDE PLS
M01648	BIT	R_3rd SPK Y HOME ENABLE
M01649	BIT	R_3rd SPK Y HOME ->
M0164B	BIT	R_3rd SPK Y START
M01656	BIT	-
M01657	BIT	-
M01658	BIT	-
M01659	BIT	-
M0165B	BIT	-
M01666	BIT	-
M01667	BIT	-
M01668	BIT	-
M01669	BIT	-
M0166B	BIT	-
M02018	BIT	-
M02019	BIT	-
M0201A	BIT	-
M0201B	BIT	-
M0201C	BIT	-
M0201D	BIT	-
M02028	BIT	-
M02029	BIT	-
M0202A	BIT	-
M0202B	BIT	-
M0202C	BIT	-
M0202D	BIT	-
M0202E	BIT	T)L_P&P Y BK OFF
M02037	BIT	-
M02038	BIT	-
M02039	BIT	-
M0203A	BIT	-
M0203B	BIT	-
M0203C	BIT	-
M0203D	BIT	-
M0203E	BIT	T)L_1st_ 03 R BK OFF
M02056	BIT	T)L_1st_ 05 Y Pos.3rd
M02057	BIT	-
M02058	BIT	-
M02059	BIT	-
M0205A	BIT	-
M0205B	BIT	-
M0205C	BIT	-
M0205D	BIT	-
M0205E	BIT	T)L_1st_ 05 Y BK OFF
M02067	BIT	-
M02068	BIT	-
M02069	BIT	-
M0206A	BIT	-
M0206B	BIT	-
M0206C	BIT	-
M0206D	BIT	-
M0206E	BIT	T)L_2nd_ 06 Y BK OFF
M02077	BIT	-
M02078	BIT	-
M02079	BIT	-
M0207A	BIT	-
M0207B	BIT	-
M0207C	BIT	-
M0207D	BIT	-
M0207E	BIT	T)L_2nd_ 07 R BK OFF
M02086	BIT	T)L_2nd_ 08 T Pos.3rd
M02088	BIT	-
M02089	BIT	-
M0208A	BIT	-
M0208B	BIT	-
M0208C	BIT	-
M0208D	BIT	-
M0208E	BIT	T)L_2nd_ 08 T BK OFF
M02098	BIT	-
M02099	BIT	-
M0209A	BIT	-
M0209B	BIT	-
M0209C	BIT	-
M0209D	BIT	-
M02108	BIT	-
M02109	BIT	-
M0210A	BIT	-
M0210B	BIT	-
M0210C	BIT	-
M0210D	BIT	-
M0210E	BIT	T)R_P&P Y BK OFF
M02117	BIT	-
M02118	BIT	-
M02119	BIT	-
M0211A	BIT	-
M0211B	BIT	-
M0211C	BIT	-
M0211D	BIT	-
M0211E	BIT	T)R_1st_11 R BK OFF
M02124	BIT	T)R_1-2 ROT R IDLE POS ->
M02125	BIT	T)R_1-2 ROT R ROT POS ->
M02126	BIT	T)R_1-2 ROT R BACK POS ->
M02127	BIT	-
M02128	BIT	-
M02129	BIT	-
M0212A	BIT	-
M0212B	BIT	-
M0212C	BIT	-
M0212D	BIT	-
M0212E	BIT	T)R_1-2 ROT R BK OFF
M02136	BIT	T)L_1st_05 Y Pos.3rd
M02137	BIT	-
M02138	BIT	-
M02139	BIT	-
M0213A	BIT	-
M0213B	BIT	-
M0213C	BIT	-
M0213D	BIT	-
M0213E	BIT	T)L_1st_05 Y BK OFF
M02147	BIT	-
M02148	BIT	-
M02149	BIT	-
M0214A	BIT	-
M0214B	BIT	-
M0214C	BIT	-
M0214D	BIT	-
M0214E	BIT	T)R_2nd_ 14 Y BK OFF
M02157	BIT	-
M02158	BIT	-
M02159	BIT	-
M0215A	BIT	-
M0215B	BIT	-
M0215C	BIT	-
M0215D	BIT	-
M0215E	BIT	T)R_2nd_ 15 R BK OFF
M02166	BIT	T)R_2nd_ 16 T Pos.3rd
M02168	BIT	-
M02169	BIT	-
M0216A	BIT	-
M0216B	BIT	-
M0216C	BIT	-
M0216D	BIT	-
M0216E	BIT	T)L_2nd_ 16 T BK OFF
M03016	BIT	-
M03017	BIT	-
M03018	BIT	-
M03019	BIT	-
M0301B	BIT	-
M0301D	BIT	-
M0301E	BIT	-
M03026	BIT	-
M03027	BIT	-
M03028	BIT	-
M03029	BIT	-
M0302B	BIT	-
M0302D	BIT	-
M0302E	BIT	-
M0302F	BIT	-
M03036	BIT	-
M03037	BIT	-
M03038	BIT	-
M03039	BIT	-
M0303B	BIT	-
M0303D	BIT	-
M0303E	BIT	-
M0303F	BIT	-
M03046	BIT	-
M03047	BIT	-
M03048	BIT	-
M03049	BIT	-
M0304B	BIT	-
M0304D	BIT	-
M0304E	BIT	-
M0304F	BIT	-
M03056	BIT	-
M03057	BIT	-
M03058	BIT	-
M03059	BIT	-
M0305B	BIT	-
M0305D	BIT	-
M0305E	BIT	-
M0305F	BIT	-
M03066	BIT	-
M03067	BIT	-
M03068	BIT	-
M03069	BIT	-
M0306B	BIT	-
M0306D	BIT	-
M0306E	BIT	-
M0306F	BIT	-
M03076	BIT	-
M03077	BIT	-
M03078	BIT	-
M03079	BIT	-
M0307B	BIT	-
M0307D	BIT	-
M0307E	BIT	-
M0307F	BIT	-
M03086	BIT	-
M03087	BIT	-
M03088	BIT	-
M03089	BIT	-
M0308B	BIT	-
M0308D	BIT	-
M0308E	BIT	-
M0308F	BIT	-
M03096	BIT	-
M03097	BIT	-
M03098	BIT	-
M03099	BIT	-
M0309B	BIT	-
M0309D	BIT	-
M0309E	BIT	-
M03106	BIT	-
M03107	BIT	-
M03108	BIT	-
M03109	BIT	-
M0310B	BIT	-
M0310D	BIT	-
M0310E	BIT	-
M0310F	BIT	-
M03116	BIT	-
M03117	BIT	-
M03118	BIT	-
M03119	BIT	-
M0311B	BIT	-
M0311D	BIT	-
M0311E	BIT	-
M0311F	BIT	-
M03126	BIT	-
M03127	BIT	-
M03128	BIT	-
M03129	BIT	-
M0312B	BIT	-
M0312D	BIT	-
M0312E	BIT	-
M0312F	BIT	-
M03136	BIT	-
M03137	BIT	-
M03138	BIT	-
M03139	BIT	-
M0313B	BIT	-
M0313D	BIT	-
M0313E	BIT	-
M0313F	BIT	-
M03146	BIT	-
M03147	BIT	-
M03148	BIT	-
M03149	BIT	-
M0314B	BIT	-
M0314D	BIT	-
M0314E	BIT	-
M0314F	BIT	-
M03156	BIT	-
M03157	BIT	-
M03158	BIT	-
M03159	BIT	-
M0315B	BIT	-
M0315D	BIT	-
M0315E	BIT	-
M0315F	BIT	-
M03166	BIT	-
M03167	BIT	-
M03168	BIT	-
M03169	BIT	-
M0316B	BIT	-
M0316D	BIT	-
M0316E	BIT	-
M0316F	BIT	-
M04016	BIT	-
M04017	BIT	-
M04018	BIT	-
M04019	BIT	-
M0401A	BIT	-
M0401B	BIT	-
M0401C	BIT	-
M0401D	BIT	-
M0401E	BIT	-
M0401F	BIT	-
M04026	BIT	-
M04027	BIT	-
M04028	BIT	-
M04029	BIT	-
M0402A	BIT	-
M0402B	BIT	-
M0402C	BIT	-
M0402D	BIT	-
M0402E	BIT	-
M0402F	BIT	-
M04036	BIT	-
M04037	BIT	-
M04038	BIT	-
M04039	BIT	-
M0403A	BIT	-
M0403B	BIT	-
M0403C	BIT	-
M0403D	BIT	-
M0403E	BIT	-
M0403F	BIT	-
M04043	BIT	-
M04044	BIT	-
M04045	BIT	-
M04046	BIT	-
M04047	BIT	-
M04048	BIT	-
M04049	BIT	-
M0404A	BIT	-
M0404B	BIT	-
M0404C	BIT	-
M0404D	BIT	-
M0404E	BIT	-
M0404F	BIT	-
M04056	BIT	-
M04057	BIT	-
M04058	BIT	-
M04059	BIT	-
M0405A	BIT	-
M0405B	BIT	-
M0405C	BIT	-
M0405D	BIT	-
M0405E	BIT	-
M0405F	BIT	-
M04066	BIT	-
M04067	BIT	-
M04068	BIT	-
M04069	BIT	-
M0406A	BIT	-
M0406B	BIT	-
M0406C	BIT	-
M0406D	BIT	-
M0406E	BIT	-
M0406F	BIT	-
M04076	BIT	-
M04077	BIT	-
M04078	BIT	-
M04079	BIT	-
M0407A	BIT	-
M0407B	BIT	-
M0407C	BIT	-
M0407D	BIT	-
M0407E	BIT	-
M0407F	BIT	-
M04086	BIT	-
M04087	BIT	-
M04088	BIT	-
M04089	BIT	-
M0408A	BIT	-
M0408B	BIT	-
M0408C	BIT	-
M0408D	BIT	-
M0408E	BIT	-
M0408F	BIT	-
M04096	BIT	-
M04097	BIT	-
M04098	BIT	-
M04099	BIT	-
M0409A	BIT	-
M0409B	BIT	-
M0409C	BIT	-
M0409D	BIT	-
M0409E	BIT	-
M0409F	BIT	-
M04106	BIT	-
M04107	BIT	-
M04108	BIT	-
M04109	BIT	-
M0410A	BIT	-
M0410B	BIT	-
M0410C	BIT	-
M0410D	BIT	-
M0410E	BIT	-
M0410F	BIT	-
M04116	BIT	-
M04117	BIT	-
M04118	BIT	-
M04119	BIT	-
M0411A	BIT	-
M0411B	BIT	-
M0411C	BIT	-
M0411D	BIT	-
M0411E	BIT	-
M0411F	BIT	-
M04123	BIT	-
M04124	BIT	-
M04125	BIT	-
M04126	BIT	-
M04127	BIT	-
M04128	BIT	-
M04129	BIT	-
M0412A	BIT	-
M0412B	BIT	-
M0412C	BIT	-
M0412D	BIT	-
M0412E	BIT	-
M0412F	BIT	-
M04136	BIT	-
M04137	BIT	-
M04138	BIT	-
M04139	BIT	-
M0413A	BIT	-
M0413B	BIT	-
M0413C	BIT	-
M0413D	BIT	-
M0413E	BIT	-
M0413F	BIT	-
M04146	BIT	-
M04147	BIT	-
M04148	BIT	-
M04149	BIT	-
M0414A	BIT	-
M0414B	BIT	-
M0414C	BIT	-
M0414D	BIT	-
M0414E	BIT	-
M0414F	BIT	-
M04156	BIT	-
M04157	BIT	-
M04158	BIT	-
M04159	BIT	-
M0415A	BIT	-
M0415B	BIT	-
M0415C	BIT	-
M0415D	BIT	-
M0415E	BIT	-
M0415F	BIT	-
M04166	BIT	-
M04167	BIT	-
M04168	BIT	-
M04169	BIT	-
M0416A	BIT	-
M0416B	BIT	-
M0416C	BIT	-
M0416D	BIT	-
M0416E	BIT	-
M0416F	BIT	-
M0062D	BIT	-
M0062E	BIT	-
M0062F	BIT	-
M00647	BIT	-
M00648	BIT	-
M00649	BIT	-
M0064B	BIT	-
M0064C	BIT	-
M0064D	BIT	-
M0064E	BIT	-
M0064F	BIT	-
M0066D	BIT	-
M0066E	BIT	-
M0067E	BIT	-
M0067F	BIT	-
M00687	BIT	-
M00688	BIT	-
M00689	BIT	-
M0068A	BIT	-
M0068B	BIT	-
M0068C	BIT	-
M0068D	BIT	-
M0068E	BIT	-
M0068F	BIT	-
M0070D	BIT	-
M0070E	BIT	-
M00727	BIT	-
M00728	BIT	-
M00729	BIT	-
M0072A	BIT	-
M0072B	BIT	-
M0072C	BIT	-
M0072D	BIT	-
M0072E	BIT	-
M0072F	BIT	-
M0073B	BIT	R_2nd MAND BTM FIX FWD/BWD SN ALARM
M0074D	BIT	-
M0074E	BIT	-
M0075E	BIT	-
M0075F	BIT	-
M00767	BIT	-
M00768	BIT	-
M00769	BIT	-
M0076A	BIT	-
M0076B	BIT	-
M0076C	BIT	-
M0076D	BIT	-
M0076E	BIT	-
M0076F	BIT	-
D01000.1	BIT	L_4th BD Z SVD RDY
D01000.4	BIT	L_4th BD Z RESET ¢¯I¡¤a
D01000.9	BIT	L_4th BD Z S4th CMD
D01000.D	BIT	L_4th BD Z DOG ¨ù¨ú¨ù¡©
D01020.1	BIT	L_P&P Y SVD RDY
D01020.4	BIT	L_P&P Y RESET ¢¯I¡¤a
D01020.9	BIT	L_P&P Y S4th CMD
D01020.D	BIT	L_P&P Y DOG ¨ù¨ú¨ù¡©
D01040.1	BIT	L_1-1 ROT R SVD RDY
D01040.4	BIT	L_1-1 ROT R RESET ¢¯I¡¤a
D01040.9	BIT	L_1-1 ROT R S4th CMD
D01040.D	BIT	L_1-1 ROT R DOG ¨ù¨ú¨ù¡©
D01060.1	BIT	L_1-2 ROT R SVD RDY
D01060.4	BIT	L_1-2 ROT R RESET ¢¯I¡¤a
D01060.9	BIT	L_1-2 ROT R S4th CMD
D01060.D	BIT	L_1-2 ROT R DOG ¨ù¨ú¨ù¡©
D01080.1	BIT	L_1st ROT Y SVD RDY
D01080.4	BIT	L_1st ROT Y RESET ¢¯I¡¤a
D01080.9	BIT	L_1st ROT Y S4th CMD
D01080.D	BIT	L_1st ROT Y DOG ¨ù¨ú¨ù¡©
D01100.1	BIT	L_3rd SPK Y SVD RDY
D01100.4	BIT	L_3rd SPK Y RESET ¢¯I¡¤a
D01100.9	BIT	L_3rd SPK Y S4th CMD
D01100.D	BIT	L_3rd SPK Y DOG ¨ù¨ú¨ù¡©
D01120.1	BIT	L_3rd ROT R SVD RDY
D01120.4	BIT	L_3rd ROT R RESET ¢¯I¡¤a
D01120.9	BIT	L_3rd ROT R STOP CMD
D01120.D	BIT	L_3rd ROT R DOG ¨ù¨ú¨ù¡©
D01140.1	BIT	L_3rd ROT Y SVD RDY
D01140.4	BIT	L_3rd ROT Y RESET ¢¯I¡¤a
D01140.9	BIT	L_3rd ROT Y STOP CMD
D01140.D	BIT	L_3rd ROT Y DOG ¨ù¨ú¨ù¡©
D01160.1	BIT	R_4th BD Z SVD RDY
D01160.4	BIT	R_4th BD Z RESET ¢¯I¡¤a
D01160.9	BIT	R_4th BD Z S4th CMD
D01160.D	BIT	R_4th BD Z DOG ¨ù¨ú¨ù¡©
D01180.1	BIT	R_P&P Y SVD RDY
D01180.4	BIT	R_P&P Y RESET ¢¯I¡¤a
D01180.9	BIT	R_P&P Y S4th CMD
D01180.D	BIT	R_P&P Y DOG ¨ù¨ú¨ù¡©
D01200.1	BIT	R_1-1 ROT R SVD RDY
D01200.4	BIT	R_1-1 ROT R RESET ¢¯I¡¤a
D01200.9	BIT	R_1-1 ROT R S4th CMD
D01200.D	BIT	R_1-1 ROT R DOG ¨ù¨ú¨ù¡©
D01220.1	BIT	R_1-2 ROT R SVD RDY
D01220.4	BIT	R_1-2 ROT R RESET ¢¯I¡¤a
D01220.9	BIT	R_1-2 ROT R S4th CMD
D01220.D	BIT	R_1-2 ROT R DOG ¨ù¨ú¨ù¡©
D01240.1	BIT	R_1st ROT Y SVD RDY
D01240.4	BIT	R_1st ROT Y RESET ¢¯I¡¤a
D01240.9	BIT	R_1st ROT Y S4th CMD
D01240.D	BIT	R_1st ROT Y DOG ¨ù¨ú¨ù¡©
D01260.1	BIT	R_3rd SPK Y SVD RDY
D01260.4	BIT	R_3rd SPK Y RESET ¢¯I¡¤a
D01260.9	BIT	R_3rd SPK Y S4th CMD
D01260.D	BIT	R_3rd SPK Y DOG ¨ù¨ú¨ù¡©
D01280.1	BIT	R_3rd ROT R SVD RDY
D01280.4	BIT	R_3rd ROT R RESET ¢¯I¡¤a
D01280.9	BIT	R_3rd ROT R STOP CMD
D01280.D	BIT	R_3rd ROT R DOG ¨ù¨ú¨ù¡©
D01300.1	BIT	R_3rd ROT Y SVD RDY
D01300.4	BIT	R_3rd ROT Y RESET ¢¯I¡¤a
D01300.9	BIT	R_3rd ROT Y STOP CMD
D01300.D	BIT	R_3rd ROT Y DOG ¨ù¨ú¨ù¡©
D02000.3	BIT	L_4th BD Z ZERO SET
D02000.8	BIT	L_4th BD Z INC POS MV
D02000.9	BIT	L_4th BD Z SPD MV
D02000.A	BIT	L_4th BD Z TRQ MV
D02000.D	BIT	L_4th BD Z A¢´Ao
D02000.F	BIT	L_4th BD Z Au¨ùO/¡Æi¨ùO
D02020.3	BIT	L_P&P Y ZERO SET
D02020.8	BIT	L_P&P Y INC POS MV
D02020.9	BIT	L_P&P Y SPD MV
D02020.A	BIT	L_P&P Y TRQ MV
D02020.D	BIT	L_P&P Y A¢´Ao
D02020.F	BIT	L_P&P Y Au¨ùO/¡Æi¨ùO
D02040.3	BIT	L_1-1 ROT R ZERO SET
D02040.8	BIT	L_1-1 ROT R INC POS MV
D02040.9	BIT	L_1-1 ROT R SPD MV
D02040.A	BIT	L_1-1 ROT R TRQ MV
D02040.D	BIT	L_1-1 ROT R A¢´Ao
D02040.F	BIT	L_1-1 ROT R Au¨ùO/¡Æi¨ùO
D02060.3	BIT	L_1-2 ROT R ZERO SET
D02060.8	BIT	L_1-2 ROT R INC POS MV
D02060.9	BIT	L_1-2 ROT R SPD MV
D02060.A	BIT	L_1-2 ROT R TRQ MV
D02060.D	BIT	L_1-2 ROT R A¢´Ao
D02060.F	BIT	L_1-2 ROT R Au¨ùO/¡Æi¨ùO
D02080.3	BIT	L_1st ROT Y ZERO SET
D02080.8	BIT	L_1st ROT Y INC POS MV
D02080.9	BIT	L_1st ROT Y SPD MV
D02080.A	BIT	L_1st ROT Y TRQ MV
D02080.D	BIT	L_1st ROT Y A¢´Ao
D02080.F	BIT	L_1st ROT Y Au¨ùO/¡Æi¨ùO
D02100.3	BIT	L_3rd SPK Y ZERO SET
D02100.8	BIT	L_3rd SPK Y INC POS MV
D02100.9	BIT	L_3rd SPK Y SPD MV
D02100.A	BIT	L_3rd SPK Y TRQ MV
D02100.D	BIT	L_3rd SPK Y A¢´Ao
D02100.F	BIT	L_3rd SPK Y Au¨ùO/¡Æi¨ùO
D02120.3	BIT	L_3rd ROT R ZERO SET
D02120.8	BIT	L_3rd ROT R INC POS MV
D02120.9	BIT	L_3rd ROT R SPD MV
D02120.A	BIT	L_3rd ROT R TRQ MV
D02120.D	BIT	L_3rd ROT R A¢´Ao
D02120.F	BIT	L_3rd ROT R Au¨ùO/¡Æi¨ùO
D02140.3	BIT	L_3rd ROT Y ZERO SET
D02140.8	BIT	L_3rd ROT Y INC POS MV
D02140.9	BIT	L_3rd ROT Y SPD MV
D02140.A	BIT	L_3rd ROT Y TRQ MV
D02140.D	BIT	L_3rd ROT Y A¢´Ao
D02140.F	BIT	L_3rd ROT Y Au¨ùO/¡Æi¨ùO
D02160.3	BIT	R_4th BD Z ZERO SET
D02160.8	BIT	R_4th BD Z INC POS MV
D02160.9	BIT	R_4th BD Z SPD MV
D02160.A	BIT	R_4th BD Z TRQ MV
D02160.D	BIT	R_4th BD Z A¢´Ao
D02160.F	BIT	R_4th BD Z Au¨ùO/¡Æi¨ùO
D02180.3	BIT	R_P&P Y ZERO SET
D02180.8	BIT	R_P&P Y INC POS MV
D02180.9	BIT	R_P&P Y SPD MV
D02180.A	BIT	R_P&P Y TRQ MV
D02180.D	BIT	R_P&P Y A¢´Ao
D02180.F	BIT	R_P&P Y Au¨ùO/¡Æi¨ùO
D02200.3	BIT	R_1-1 ROT R ZERO SET
D02200.8	BIT	R_1-1 ROT R INC POS MV
D02200.9	BIT	R_1-1 ROT R SPD MV
D02200.A	BIT	R_1-1 ROT R TRQ MV
D02200.D	BIT	R_1-1 ROT R A¢´Ao
D02200.F	BIT	R_1-1 ROT R Au¨ùO/¡Æi¨ùO
D02220.3	BIT	R_1-2 ROT R ZERO SET
D02220.8	BIT	R_1-2 ROT R INC POS MV
D02220.9	BIT	R_1-2 ROT R SPD MV
D02220.A	BIT	R_1-2 ROT R TRQ MV
D02220.D	BIT	R_1-2 ROT R A¢´Ao
D02220.F	BIT	R_1-2 ROT R Au¨ùO/¡Æi¨ùO
D02240.3	BIT	R_1st ROT Y ZERO SET
D02240.8	BIT	R_1st ROT Y INC POS MV
D02240.9	BIT	R_1st ROT Y SPD MV
D02240.A	BIT	R_1st ROT Y TRQ MV
D02240.D	BIT	R_1st ROT Y A¢´Ao
D02240.F	BIT	R_1st ROT Y Au¨ùO/¡Æi¨ùO
D02260.3	BIT	R_3rd SPK Y ZERO SET
D02260.8	BIT	R_3rd SPK Y INC POS MV
D02260.9	BIT	R_3rd SPK Y SPD MV
D02260.A	BIT	R_3rd SPK Y TRQ MV
D02260.D	BIT	R_3rd SPK Y A¢´Ao
D02260.F	BIT	R_3rd SPK Y Au¨ùO/¡Æi¨ùO
D02280.3	BIT	R_3rd ROT R ZERO SET
D02280.8	BIT	R_3rd ROT R INC POS MV
D02280.9	BIT	R_3rd ROT R SPD MV
D02280.A	BIT	R_3rd ROT R TRQ MV
D02280.D	BIT	R_3rd ROT R A¢´Ao
D02280.F	BIT	R_3rd ROT R Au¨ùO/¡Æi¨ùO
D02300.3	BIT	R_3rd ROT Y ZERO SET
D02300.8	BIT	R_3rd ROT Y INC POS MV
D02300.9	BIT	R_3rd ROT Y SPD MV
D02300.A	BIT	R_3rd ROT Y TRQ MV
D02300.D	BIT	R_3rd ROT Y A¢´Ao
D02300.F	BIT	R_3rd ROT Y Au¨ùO/¡Æi¨ùO
D02000	WORD	-
D02001	WORD	-
D02003	WORD	-
D02005	WORD	-
D02006	WORD	-
D02007	WORD	-
D02009	WORD	-
D02010	WORD	L_4th BD Z A¢Ò¡¾¡¿¡Æi¨ùO
D02011	WORD	-
D02013	WORD	-
D02015	WORD	-
D02023	WORD	-
D02025	WORD	-
D02026	WORD	-
D02027	WORD	-
D02029	WORD	-
D02030	WORD	L_P&P Y A¢Ò¡¾¡¿¡Æi¨ùO
D02031	WORD	-
D02033	WORD	-
D02035	WORD	-
D02040	WORD	-
D02041	WORD	-
D02043	WORD	-
D02045	WORD	-
D02046	WORD	-
D02047	WORD	-
D02049	WORD	-
D02050	WORD	L_1st ROT R A¢Ò¡¾¡¿¡Æi¨ùO
D02051	WORD	-
D02053	WORD	-
D02055	WORD	-
D02060	WORD	-
D02061	WORD	-
D02063	WORD	-
D02065	WORD	-
D02066	WORD	-
D02067	WORD	-
D02069	WORD	-
D02070	WORD	L_1st ROT X A¢Ò¡¾¡¿¡Æi¨ùO
D02071	WORD	-
D02073	WORD	-
D02075	WORD	-
D02080	WORD	-
D02081	WORD	-
D02083	WORD	-
D02085	WORD	-
D02086	WORD	-
D02087	WORD	-
D02089	WORD	-
D02090	WORD	L_2nd ROT R A¢Ò¡¾¡¿¡Æi¨ùO
D02091	WORD	-
D02093	WORD	-
D02095	WORD	-
D02100	WORD	-
D02101	WORD	-
D02103	WORD	-
D02105	WORD	-
D02106	WORD	-
D02107	WORD	-
D02109	WORD	-
D02110	WORD	L_2nd ROT Y A¢Ò¡¾¡¿¡Æi¨ùO
D02111	WORD	-
D02113	WORD	-
D02115	WORD	-
D02120	WORD	-
D02121	WORD	-
D02123	WORD	-
D02125	WORD	-
D02126	WORD	-
D02127	WORD	-
D02129	WORD	-
D02130	WORD	L_3rd ROT R A¢Ò¡¾¡¿¡Æi¨ùO
D02131	WORD	-
D02133	WORD	-
D02135	WORD	-
D02140	WORD	-
D02141	WORD	-
D02143	WORD	-
D02145	WORD	-
D02146	WORD	-
D02147	WORD	-
D02149	WORD	-
D02150	WORD	L_3rd ROT Y A¢Ò¡¾¡¿¡Æi¨ùO
D02151	WORD	-
D02153	WORD	-
D02155	WORD	-
D02160	WORD	-
D02161	WORD	-
D02163	WORD	-
D02165	WORD	-
D02166	WORD	-
D02167	WORD	-
D02169	WORD	-
D02170	WORD	R_4th BD Z A¢Ò¡¾¡¿¡Æi¨ùO
D02171	WORD	-
D02173	WORD	-
D02175	WORD	-
D02180	WORD	-
D02181	WORD	-
D02183	WORD	-
D02185	WORD	-
D02186	WORD	-
D02187	WORD	-
D02189	WORD	-
D02190	WORD	R_P&P Y A¢Ò¡¾¡¿¡Æi¨ùO
D02191	WORD	-
D02193	WORD	-
D02195	WORD	-
D02200	WORD	-
D02201	WORD	-
D02203	WORD	-
D02205	WORD	-
D02206	WORD	-
D02207	WORD	-
D02209	WORD	-
D02210	WORD	R_1st ROT R A¢Ò¡¾¡¿¡Æi¨ùO
D02211	WORD	-
D02213	WORD	-
D02215	WORD	-
D02220	WORD	-
D02221	WORD	-
D02223	WORD	-
D02225	WORD	-
D02226	WORD	-
D02227	WORD	-
D02229	WORD	-
D02230	WORD	R_1st ROT X A¢Ò¡¾¡¿¡Æi¨ùO
D02231	WORD	-
D02233	WORD	-
D02235	WORD	-
D02240	WORD	-
D02241	WORD	-
D02243	WORD	-
D02245	WORD	-
D02246	WORD	-
D02247	WORD	-
D02249	WORD	-
D02250	WORD	R_2nd ROT R A¢Ò¡¾¡¿¡Æi¨ùO
D02251	WORD	-
D02253	WORD	-
D02255	WORD	-
D02260	WORD	-
D02261	WORD	-
D02263	WORD	-
D02265	WORD	-
D02266	WORD	-
D02267	WORD	-
D02269	WORD	-
D02270	WORD	R_2nd ROT Y A¢Ò¡¾¡¿¡Æi¨ùO
D02271	WORD	-
D02273	WORD	-
D02275	WORD	-
D02280	WORD	-
D02281	WORD	-
D02283	WORD	-
D02285	WORD	-
D02286	WORD	-
D02287	WORD	-
D02289	WORD	-
D02290	WORD	R_3rd ROT R A¢Ò¡¾¡¿¡Æi¨ùO
D02291	WORD	-
D02293	WORD	-
D02295	WORD	-
D02300	WORD	-
D02301	WORD	-
D02303	WORD	-
D02305	WORD	-
D02306	WORD	-
D02307	WORD	-
D02309	WORD	-
D02310	WORD	R_3rd ROT Y A¢Ò¡¾¡¿¡Æi¨ùO
D02311	WORD	-
D02313	WORD	-
D02315	WORD	-
P00018	BIT	-
P00019	BIT	-
P0002F	BIT	-
P00031	BIT	-
P0003B	BIT	-
P00041	BIT	-
P0004F	BIT	-
P0006F	BIT	-
P00071	BIT	-
P0007B	BIT	-
P00081	BIT	-
P00096	BIT	L_1st CLAMP Z BRAKE
P00106	BIT	R_1st CLAMP Z BRAKE
P0011B	BIT	-
P0013D	BIT	-
P0013E	BIT	-
P0013F	BIT	-
P0014A	BIT	-
P0014B	BIT	-
P0014F	BIT	-
P0015E	BIT	-
P0016F	BIT	-
T0293	BIT/WORD	RT_P&P UP
T0283	BIT/WORD	LF_P&P UP
M10642	BIT	L_2nd MAND BTM FIX FWD
M10644	BIT	L_2nd MAND SPANKING FWD
M10650	BIT	L_2nd MAND FWD
T0383	BIT/WORD	L_2nd MAND BTM SN ALARM
T0384	BIT/WORD	L_2nd MAND BTM FIX FWD/BWD SN ALARM
M0065B	BIT	L_2nd MAND BTM FIX FWD/BWD SN ALARM
T0385	BIT/WORD	L_2nd MAND SPANKING FWD/BWD SN ALARM
T0386	BIT/WORD	L_2nd MAND FWD/BWD SN ALARM
T0850	BIT/WORD	R_IN BUFFER DIE LD/PP SN ALARM
T0583	BIT/WORD	R_2nd MAND BTM SN ALARM
T0584	BIT/WORD	R_2nd MAND BTM FIX FWD/BWD SN ALARM
T0585	BIT/WORD	R_2nd MAND SPANKING FWD/BWD SN ALARM
T0586	BIT/WORD	R_2nd MAND FWD/BWD SN ALARM
M13300	BIT	T)R_2nd ROT R IDLE POS PLS
M13302	BIT	T)R_2nd ROT R IDLE POS ->
M13304	BIT	T)R_2nd ROT R ROT POS PLS
M13306	BIT	T)R_2nd ROT R ROT POS ->
M13308	BIT	T)R_2nd ROT R BACK POS PLS
M1330A	BIT	T)R_2nd ROT R BACK POS ->
M14694	BIT	R_4th TOOL AUAc ¡Æ¢®A¢ç¡Æ¡§
M1469F	BIT	R_4th TOOL AUAc ¨ú©ª¨úiAu
P00037	BIT	-
P00038	BIT	-
P00039	BIT	-
P0003A	BIT	-
P0003C	BIT	-
P00077	BIT	-
P00078	BIT	-
P00079	BIT	-
P0007A	BIT	-
P0007C	BIT	-
P0014D	BIT	-
P0001A	BIT	-
P0001B	BIT	-
P0001C	BIT	-
P0003D	BIT	-
P0003E	BIT	-
P0003F	BIT	-
P0007D	BIT	-
P0007E	BIT	-
P0007F	BIT	-
P0014E	BIT	-
P0015F	BIT	-
M01676	BIT	L_3rd BD Z SPD MV PLS
M01677	BIT	L_3rd BD Z OVERRIDE PLS
M01678	BIT	L_3rd BD Z HOME ENABLE
M01679	BIT	L_3rd BD Z HOME ->
M0167B	BIT	L_3rd BD Z START
M01686	BIT	R_3rd BD Z SPD MV PLS
M01687	BIT	R_3rd BD Z OVERRIDE PLS
M01688	BIT	R_3rd BD Z HOME ENABLE
M01689	BIT	R_3rd BD Z HOME ->
M0168B	BIT	R_3rd BD Z START
M02178	BIT	-
M02179	BIT	-
M0217A	BIT	-
M0217B	BIT	-
M0217C	BIT	-
M0217D	BIT	-
M0217E	BIT	T)L_3rd_17 Z BK OFF
M02188	BIT	-
M02189	BIT	-
M0218A	BIT	-
M0218B	BIT	-
M0218C	BIT	-
M0218D	BIT	-
M0218E	BIT	T)R_3rd_18 Z BK OFF
M03176	BIT	-
M03177	BIT	-
M03178	BIT	-
M03179	BIT	-
M0317B	BIT	-
M0317D	BIT	-
M0317E	BIT	-
M03186	BIT	-
M03187	BIT	-
M03188	BIT	-
M03189	BIT	-
M0318B	BIT	-
M0318D	BIT	-
M0318E	BIT	-
M04176	BIT	-
M04177	BIT	-
M04178	BIT	-
M04179	BIT	-
M0417A	BIT	-
M0417B	BIT	-
M0417C	BIT	-
M0417D	BIT	-
M0417E	BIT	-
M0417F	BIT	-
M04186	BIT	-
M04187	BIT	-
M04188	BIT	-
M04189	BIT	-
M0418A	BIT	-
M0418B	BIT	-
M0418C	BIT	-
M0418D	BIT	-
M0418E	BIT	-
M0418F	BIT	-
M0077B	BIT	-
M0077C	BIT	-
M0077D	BIT	-
M0077E	BIT	-
M0078B	BIT	-
M0078C	BIT	-
M0078D	BIT	-
M0078E	BIT	-
D01320.1	BIT	L_3rd BD Z SVD RDY
D01320.4	BIT	L_3rd BD Z RESET ¢¯I¡¤a
D01320.9	BIT	L_3rd BD Z S4th CMD
D01320.D	BIT	L_3rd BD Z DOG ¨ù¨ú¨ù¡©
D01340.1	BIT	R_3rd BD Z SVD RDY
D01340.4	BIT	R_3rd BD Z RESET ¢¯I¡¤a
D01340.9	BIT	R_3rd BD Z S4th CMD
D01340.D	BIT	R_3rd BD Z DOG ¨ù¨ú¨ù¡©
D02320.3	BIT	L_3rd BD Z ZERO SET
D02320.8	BIT	L_3rd BD Z INC POS MV
D02320.9	BIT	L_3rd BD Z SPD MV
D02320.A	BIT	L_3rd BD Z TRQ MV
D02320.D	BIT	L_3rd BD Z A¢´Ao
D02320.F	BIT	L_3rd BD Z Au¨ùO/¡Æi¨ùO
D02340.3	BIT	R_3rd BD Z ZERO SET
D02340.8	BIT	R_3rd BD Z INC POS MV
D02340.9	BIT	R_3rd BD Z SPD MV
D02340.A	BIT	R_3rd BD Z TRQ MV
D02340.D	BIT	R_3rd BD Z A¢´Ao
D02340.F	BIT	R_3rd BD Z Au¨ùO/¡Æi¨ùO
D02320	WORD	-
D02321	WORD	-
D02323	WORD	-
D02325	WORD	-
D02326	WORD	-
D02327	WORD	-
D02329	WORD	-
D02330	WORD	L_3rd BD Z A¢Ò¡¾¡¿¡Æi¨ùO
D02331	WORD	-
D02333	WORD	-
D02335	WORD	-
D02340	WORD	-
D02341	WORD	-
D02343	WORD	-
D02345	WORD	-
D02346	WORD	-
D02347	WORD	-
D02349	WORD	-
D02350	WORD	R_3rd BD Z A¢Ò¡¾¡¿¡Æi¨ùO
D02351	WORD	-
D02353	WORD	-
D02355	WORD	-
M1057B	BIT	L_2nd TOP FIX CLAMP UP
M1057C	BIT	L_2nd TOP LATCH CLAMP UP
M1057D	BIT	L_2nd ROT R IDLE POS
M1057E	BIT	L_2nd ROT Y MANDREL POS
M1307B	BIT	R_2nd TOP FIX CLAMP UP
M1307C	BIT	R_2nd TOP LATCH CLAMP UP
M1307D	BIT	R_2nd ROT R IDLE POS
M1307E	BIT	R_2nd ROT Y MANDREL POS
M11066	BIT	-
M11067	BIT	-
M1107B	BIT	L_3rd BTM ROT R RECEIVE POS
M13566	BIT	-
M13567	BIT	-
M1357B	BIT	R_3rd BTM ROT R RECEIVE POS
M1107C	BIT	L_3rd BTM ROT R WORK POS
M1107D	BIT	L_3rd TOP CLAMP FWD/BWD SENSOR
M1357C	BIT	R_3rd BTM ROT R WORK POS
M1357D	BIT	R_3rd TOP CLAMP FWD/BWD SENSOR
M11370	BIT	T)L_3rd SPANKING FWD/BWD PLS
M11372	BIT	T)L_3rd SPANKING BWD
M11374	BIT	T)L_3rd SPANKING FWD
M13870	BIT	T)R_3rd SPANKING FWD/BWD PLS
M13872	BIT	T)R_3rd SPANKING BWD
M13874	BIT	T)R_3rd SPANKING FWD
M02087	BIT	-
M1132C	BIT	T)L_3rd ROT Y IDLE POS PLS
M1132E	BIT	T)L_3rd ROT Y IDLE POS ->
M02167	BIT	-
M1382C	BIT	T)R_3rd ROT Y IDLE POS PLS
M1382E	BIT	T)R_3rd ROT Y IDLE POS ->
M1307F	BIT	R_2nd MANDREL BACKWARD
M1057F	BIT	L_2nd MANDREL BACKWARD
D06950	WORD	LOT NO + RIGHT
M0026A	BIT	10_AU¥ì¢¯ STEP END PLS
M00260	BIT	RIGHT CYCLE TIME LOG
D03045.D	BIT	X1862
M00379	BIT	MES NG PLS
P00030	BIT	-
P00040	BIT	-
P00070	BIT	-
P00080	BIT	-
T0763	BIT/WORD	-
M00787	BIT	R_3rd MAND DIE ALIGN FWD/BWD SN ALARM
D03045.B	BIT	ZAa ¢¬OAu ¡ío¨öA
D37021	WORD	'¢¯u' ¥ì¡ÍAIAI
D37022	WORD	'AI' ¥ì¡ÍAIAI
D37023	WORD	'¨öA' ¥ì¡ÍAIAI
D37024	WORD	'¨¬¨¢' ¥ì¡ÍAIAI
D37025	WORD	'AE' ¥ì¡ÍAIAI
M08532	BIT	LOT IN LAMP
D03045.5	BIT	©öeAa ¨ù¨ú¨ù¡© ¡íc¢¯e ¨úECO
M0077F	BIT	L_3rd OVERLOAD ALARM.
D01332	WORD	L_3rd Z OVERLOAD
M0078F	BIT	R_3rd OVERLOAD ALARM.
D01352	WORD	R_3rd Z OVERLOAD
D04868	WORD	R_3rd Z OVERLOAD LIMIT
D04768	WORD	L_3rd Z OVERLOAD LIMIT
T0952	BIT/WORD	R_FRONT SAFETY SENSOR
T0953	BIT/WORD	R_REAR SAFETY SENSOR
T0323	BIT/WORD	L_1st CLP Z DN POS
T0324	BIT/WORD	R_1st CLP Z DN POS
M10067	BIT	-
M12567	BIT	-
M10640	BIT	L_2nd DIE FPCB ALIGN FWD
M10641	BIT	L_2nd DIE FPCB ALIGN BWD
M11160	BIT	L_3rd TOP DOWN
M0074C	BIT	R_3rd TOP UP/DOWN SN ALARM
M13660	BIT	R_3rd TOP DOWN
M11150	BIT	L_3rd SUPPORT DOWN
M11065	BIT	-
M11152	BIT	L_3rd SUPPORT UP
M00778	BIT	L_3rd SUPPORT UP SN ALARM
M10310	BIT	T)L_3rd BD Z UP POS ->
M10312	BIT	T)L_3rd BD Z UP POS ->
M10314	BIT	T)L_3rd BD Z CENTER POS ->
M10316	BIT	T)L_3rd BD Z CENTER POS ->
M10318	BIT	T)L_3rd BD Z BENDING POS ->
M1031A	BIT	T)L_3rd BD Z BENDING POS ->
P00067	BIT	-
M13650	BIT	R_3rd SUPPORT DOWN
M00788	BIT	R_3rd SUPPORT UP SN ALARM
M13652	BIT	R_3rd SUPPORT UP
D19200.0	BIT	fr LOADING
D19200.1	BIT	fr LOADING
D19600.0	BIT	fr UNLOADING
D19201.F	BIT	LD-SV-DATA MOVE-REQ
D19401.F	BIT	LD SV DATA ©ö¨­¡¾aOK
D19201.0	BIT	LD-BUFF HOLD-REQ
D19201.2	BIT	LOAD OK
D19402.0	BIT	LOAD STOP
D19402.1	BIT	LOAD REQ
D19402.2	BIT	BUFF HOLD ACK
D19402.4	BIT	LOAD OK ACK
D19402.3	BIT	IN-BUFF VAC ON
P00068	BIT	R-IN-BUFF ALIGN UP
P00069	BIT	R-IN-BUFF ALIGN DN
P0006C	BIT	R-IN-BUFF ALIGN FWD
P00104	BIT	R-IN-BUFF ALGN-UP
D19201.1	BIT	LDER)VAC REQ
D19601.0	BIT	OUT-BUFF HOLD REQ
D19601.2	BIT	UNLOAD OK
D19802.1	BIT	UNLOAD REQ
D19802.2	BIT	OUT-BUFF HOLD ACK
D19802.3	BIT	OUT-BUFF VAC OFF
D19802.4	BIT	UNLOAD OK ACK
D19601.1	BIT	UNLD VAC OFF REQ
M02450	BIT	R-IN-BUF ALIGN-CYC
M02455	BIT	R-IN-BUFF ALIGN_ed
D19601.F	BIT	UNLD-SVDATA MOVE-REQ
D19600.1	BIT	UNLOADING [ON]
D19400.0	BIT	to LOADING
D19800.0	BIT	to UNLOADING
D19801.F	BIT	UNLD SVDATA ©ö¨­¡¾aOK
D19400.A	BIT	AUTO RUN
D19400.B	BIT	STOP
D19400.C	BIT	ALARM
D19800.A	BIT	AUTO RUN
D19800.B	BIT	STOP
D19800.C	BIT	ALARM
D19400.2	BIT	START
D19400.3	BIT	STOP
D19400.4	BIT	RESET
D19400.5	BIT	INITIAL
D19800.2	BIT	START
D19800.3	BIT	STOP
D19800.4	BIT	RESET
D19800.5	BIT	INITIAL
D19402.A	BIT	DEV CHG
D19402.B	BIT	DEV COPY
D19802.A	BIT	DEV CHG
D19802.B	BIT	DEV COPY
D19601.A	BIT	DEV CHG ACK
D19601.B	BIT	DEV CHG NAK
D19601.C	BIT	DEV COPY ACK
D19601.D	BIT	DEV COPY NAK
D19400.9	BIT	DRY RUN
D19800.9	BIT	DRY RUN
D19201.A	BIT	DEV CHG ACK
D19201.B	BIT	DEV CHG NAK
D19201.C	BIT	DEV COPY ACK
D19201.D	BIT	DEV COPY NAK
D19204.C	BIT	LDER_Y BUFF-POS
D19208.A	BIT	LDER-Y PAD-UP
D19608.A	BIT	UNLDER-Y PAD-UP
D19604.C	BIT	UNLDER-Y BUFF-POS
M01102	BIT	¢¯¨­AE ¨öAAU ¨ö¨¬A¡×A¢®¢¬| ¢¥¡©¡¤? AO¨ù¨ù¢¯a
M01107	BIT	¨öIAIA¡þ ¢¯iAuA©¬...
M0110A	BIT	¢¯A¢¬¡ÍAE ¨öAAU ¨ö¨¬A¡×A¢®¢¬| ¢¥¡©¡¤? AO¨ù¨ù¢¯a
M01160	BIT	1160.[AoAO¡¤I¢¥o] AoAO ¢¯¢´¢¬¢ç¨¬¡ÌAIAI ZAa ¢¯©ªA¢® ¨¬©ö¡¾IA©¬¢®|
M01161	BIT	1161.[AoAO¡¤I¢¥o] AoAO 1A¡À CC¢¥o XAa ¢¯©ªA¢® ¨¬©ö¡¾IA©¬¢®|
M01162	BIT	1162.[AoAO¡¤I¢¥o] AoAO 2A¡À CC¢¥o XAa ¢¯©ªA¢® ¨¬©ö¡¾IA©¬¢®|
M01163	BIT	1163.[AoAO¡¤I¢¥o] AoAO AUAc CCA¢¯ YAa ¢¯©ªA¢® ¨¬©ö¡¾IA©¬¢®|
M01164	BIT	1164.[AoAO¡¤I¢¥o]
M01165	BIT	1165.[AoAO¡¤I¢¥o]
M01166	BIT	1166.[AoAO¡¤I¢¥o]
M01167	BIT	1167.[AoAO¡¤I¢¥o]
M01168	BIT	1168.[AoAO¡¤I¢¥o]
M01169	BIT	1169.[AoAO¡¤I¢¥o]
M0116A	BIT	116A.[AoAO¡¤I¢¥o]
M0116B	BIT	116B.[AoAO¡¤I¢¥o]
M0116C	BIT	116C.[AoAO¡¤I¢¥o]
M0116D	BIT	116D.[AoAO¡¤I¢¥o]
M0116E	BIT	116E.[AoAO¡¤I¢¥o]
M0116F	BIT	116F.[AoAO¡¤I¢¥o]
M01170	BIT	1170.[AoAO¡¤I¢¥o]
M01171	BIT	1171.[AoAO¡¤I¢¥o]
M01172	BIT	1172.[AoAO¡¤I¢¥o]
M01173	BIT	1173.[AoAO¡¤I¢¥o]
M01174	BIT	1174.[AoAO¡¤I¢¥o]
M01175	BIT	1175.[AoAO¡¤I¢¥o]
M01176	BIT	1176.[AoAO¡¤I¢¥o]
M01177	BIT	1177.[AoAO¡¤I¢¥o]
M01178	BIT	1178.[AoAO¡¤I¢¥o]
M01179	BIT	1179.[AoAO¡¤I¢¥o]
M0117A	BIT	117A.[AoAO¡¤I¢¥o]
M0117B	BIT	117B.[AoAO¡¤I¢¥o]
M0117C	BIT	117C.[AoAO¡¤I¢¥o]
M0117D	BIT	117D.[AoAO¡¤I¢¥o]
M0117E	BIT	117E.[AoAO¡¤I¢¥o]
M0117F	BIT	117F.[AoAO¡¤I¢¥o]
M01180	BIT	1180.[©öeAa¡¤I¢¥o] AoAO ¢¯¢´¢¬¢ç¨¬¡ÌAIAI ZAa ¢¯©ªA¢® ¨¬©ö¡¾IA©¬¢®|
M01181	BIT	1181.[©öeAa¡¤I¢¥o] AoAO 1A¡À CC¢¥o XAa ¢¯©ªA¢® ¨¬©ö¡¾IA©¬¢®|
M01182	BIT	1182.[©öeAa¡¤I¢¥o] AoAO 2A¡À CC¢¥o XAa ¢¯©ªA¢® ¨¬©ö¡¾IA©¬¢®|
M01183	BIT	1183.[©öeAa¡¤I¢¥o] AoAO AUAc CCA¢¯ YAa ¢¯©ªA¢® ¨¬©ö¡¾IA©¬¢®|
M01184	BIT	1184.[©öeAa¡¤I¢¥o]
M01185	BIT	1185.[©öeAa¡¤I¢¥o]
M01186	BIT	1186.[©öeAa¡¤I¢¥o]
M01187	BIT	1187.[©öeAa¡¤I¢¥o]
M01188	BIT	1188.[©öeAa¡¤I¢¥o]
M01189	BIT	1189.[©öeAa¡¤I¢¥o]
M0118A	BIT	118A.[©öeAa¡¤I¢¥o]
M0118B	BIT	118B.[©öeAa¡¤I¢¥o]
M0118C	BIT	118C.[©öeAa¡¤I¢¥o]
M0118D	BIT	118D.[©öeAa¡¤I¢¥o]
M0118E	BIT	118E.[©öeAa¡¤I¢¥o]
M0118F	BIT	118F.[©öeAa¡¤I¢¥o]
M01190	BIT	1190.[©öeAa¡¤I¢¥o]
M01191	BIT	1191.[©öeAa¡¤I¢¥o]
M01192	BIT	1192.[©öeAa¡¤I¢¥o]
M01193	BIT	1193.[©öeAa¡¤I¢¥o]
M01194	BIT	1194.[©öeAa¡¤I¢¥o]
M01195	BIT	1195.[©öeAa¡¤I¢¥o]
M01196	BIT	1196.[©öeAa¡¤I¢¥o]
M01197	BIT	1197.[©öeAa¡¤I¢¥o]
M01198	BIT	1198.[©öeAa¡¤I¢¥o]
M01199	BIT	1199.[©öeAa¡¤I¢¥o]
M0119A	BIT	119A.[©öeAa¡¤I¢¥o]
M0119B	BIT	119B.[©öeAa¡¤I¢¥o]
M0119C	BIT	119C.[©öeAa¡¤I¢¥o]
M0119D	BIT	119D.[©öeAa¡¤I¢¥o]
M0119E	BIT	119E.[©öeAa¡¤I¢¥o]
M0119F	BIT	119F.[©öeAa¡¤I¢¥o]
M00940	BIT	940.[AoAO¡¤I¢¥o] ¨¬n¡íoA¢´Ao
M00942	BIT	942.[AoAO¡¤I¢¥o] AoAO¨¬I ¨úEAu ¨ù¨ú¨ù¡© ¡Æ¡§Ao¥ìE.
M00943	BIT	943.[AoAO¡¤I¢¥o] ©öeAa¨¬I ¨úEAu ¨ù¨ú¨ù¡© ¡Æ¡§Ao¥ìE.
M00944	BIT	944.[AoAO¡¤I¢¥o] AoAO¨¬I Au¢¬e ¨úEAu©ö¢ç ¢¯¡©¢¬©÷.
M00945	BIT	945.[AoAO¡¤I¢¥o] AoAO¨¬I ¢¯¡¤¢¬e ¨úEAu©ö¢ç ¢¯¡©¢¬©÷.
M00946	BIT	946.[AoAO¡¤I¢¥o] ©öeAa¨¬I Au¢¬e ¨úEAu©ö¢ç ¢¯¡©¢¬©÷.
M00947	BIT	947.[AoAO¡¤I¢¥o] 
M00948	BIT	948.[AoAO¡¤I¢¥o] 
M00949	BIT	949.[AoAO¡¤I¢¥o] AoAO ¢¯¢´¢¬¢ç¨¬¡ÌAIAI ZAa ¢¯©ªA¢®¨¬©ö¡¾I ©öI ¢¯I¡¤a.
M0094A	BIT	94A.[AoAO¡¤I¢¥o] AoAO ¢¯¢´¢¬¢ç¨¬¡ÌAIAI ZAa A¢´¡ío A¡×A¢®¡Æ¢® ¨ú¨¡¢¥O.
M0094B	BIT	94B.[AoAO¡¤I¢¥o] AoAO ¢¯¢´¢¬¢ç¨¬¡ÌAIAI ZAa ¨ù¡©¨¬¢¬ ¥ìa¢ÒoAI©öo ¢¯¢®¡¤?©ö©¬¡íy. ¢¯¢®¡¤?AU¥ìa E¢çAI©öU¢Ò¡À.
M0094C	BIT	94C.[AoAO¡¤I¢¥o] AoAO ¢¯¢´¢¬¢ç¨¬¡ÌAIAI ZAoAO ¢¯¢´¢¬¢ç¨¬¡ÌAIAI ZAa ¨ù¡©¨¬¢¬¢¬©£AI AI¥ì¢¯CIAo ¨úEA¨ö.
M0094D	BIT	94D.[AoAO¡¤I¢¥o] AoAO ¢¯¢´¢¬¢ç¨¬¡ÌAIAI ZAoAO ¢¯¢´¢¬¢ç¨¬¡ÌAIAI ZAa ¨ù¡©¨¬¢¬¢¬©£AI +¢¬¢ç©öI¨¡¢ç.
M0094E	BIT	94E.[AoAO¡¤I¢¥o] AoAO ¢¯¢´¢¬¢ç¨¬¡ÌAIAI ZAa ¨ù¡©¨¬¢¬¢¬©£AI -¢¬¢ç©öI¨¡¢ç.
M0094F	BIT	94F.[AoAO¡¤I¢¥o] AoAO ¢¯¢´¢¬¢ç¨¬¡ÌAIAI ZAa ¨ù¡©¨¬¢¬ ¢¯ACA.
M00950	BIT	950.[AoAO¡¤I¢¥o] AoAO ¨ù¡©¨¡¡À¨¡¢ç1 ¢¯¡©¢¬©÷/¢¥YEu ¨ù¨ú¨ù¡© ¨úE¢Ò¡À.
M00951	BIT	951.[AoAO¡¤I¢¥o] AoAO ¨ù¡©¨¡¡À¨¡¢ç2 ¢¯¡©¢¬©÷/¢¥YEu ¨ù¨ú¨ù¡© ¨úE¢Ò¡À.
M00952	BIT	952.[AoAO¡¤I¢¥o] AoAO ¨¡¢ç¡¤©öAI ¨¬¨¢¢¬¢ç1 ¢¯¡©¢¬©÷/¢¥YEu ¨ù¨ú¨ù¡© ¨úE¢Ò¡À.
M00953	BIT	953.[AoAO¡¤I¢¥o] AoAO ¨¡¢ç¡¤©öAI ¨¬¨¢¢¬¢ç2 ¢¯¡©¢¬©÷/¢¥YEu ¨ù¨ú¨ù¡© ¨úE¢Ò¡À.
M00954	BIT	954.[AoAO¡¤I¢¥o] AoAO ¨¡¢ç¡¤©öAI ©öeAa ¡ío¨öA/CI¡Æ¡© ¨ù¨ú¨ù¡© ¨úE¢Ò¡À.
M00955	BIT	955.[AoAO¡¤I¢¥o] AoAO ¨¡¢ç¡¤©öAI ¢¯¢´¢¬¢ç¨¬¡ÌAIAI ¢¯¥ì¢¯¨£ ¡¤©öAIA¡× ¨úEA©ª ¨¬O¡¤¢ç.
M00956	BIT	956.[AoAO¡¤I¢¥o] AoAO ¢¯¢´¢¬¢ç¨¬¡ÌAIAI ¡ío¨öA ¡Æ¢®¢¥E ¨ù¨ú¨ù¡© ¨úE¢Ò¡À.
M00957	BIT	957.[AoAO¡¤I¢¥o] AoAO ¢¬¢çCA¨¡¢ç ¡ío¨öA ¡Æ¢®¢¥E ¨ù¨ú¨ù¡© ¨úE¢Ò¡À.
M00958	BIT	958.[AoAO¡¤I¢¥o] AoAO AU¨ú¡À ¢¯I¡¤a ¨¡¢ç¡¤©öAI ¡Æ¢®¥ì©¡Au.
M00959	BIT	959.[AoAO¡¤I¢¥o] AoAO 1A¡À CC¢¥o XAa ¢¯©ªA¢®¨¬©ö¡¾I ©öI ¢¯I¡¤a.
M0095A	BIT	95A.[AoAO¡¤I¢¥o] AoAO 1A¡À CC¢¥o XAa A¢´¡ío A¡×A¢®¡Æ¢® ¨ú¨¡¢¥O.
M0095B	BIT	95B.[AoAO¡¤I¢¥o] AoAO 1A¡À CC¢¥o XAa ¨ù¡©¨¬¢¬ ¥ìa¢ÒoAI©öo ¢¯¢®¡¤?©ö©¬¡íy. ¢¯¢®¡¤?AU¥ìa E¢çAI©öU¢Ò¡À.
M0095C	BIT	95C.[AoAO¡¤I¢¥o] AoAO 1A¡À CC¢¥o XAa ¨ù¡©¨¬¢¬¢¬©£AI AI¥ì¢¯CIAo ¨úEA¨ö.
M0095D	BIT	95D.[AoAO¡¤I¢¥o] AoAO 1A¡À CC¢¥o XAa ¨ù¡©¨¬¢¬¢¬©£AI +¢¬¢ç©öI¨¡¢ç.
M0095E	BIT	95E.[AoAO¡¤I¢¥o] AoAO 1A¡À CC¢¥o XAa ¨ù¡©¨¬¢¬¢¬©£AI -¢¬¢ç©öI¨¡¢ç.
M0095F	BIT	95F.[AoAO¡¤I¢¥o] AoAO 1A¡À CC¢¥o XAa ¨ù¡©¨¬¢¬ ¢¯ACA.
M00960	BIT	960.[AoAO¡¤I¢¥o] AoAO 1A¡À CC¢¥o A¡þ¡¤¡ÍCA ¢¯¡©¢¬©÷/¢¥YEu ¨ù¨ú¨ù¡© ¨úE¢Ò¡À.
M00961	BIT	961.[AoAO¡¤I¢¥o] AoAO ¨¡¢ç¡¤©öAI ¢¯¡¤ A¡þ¡¤¡ÍCA ¢¯¡©¢¬©÷/¢¥YEu ¨ù¨ú¨ù¡© ¨úE¢Ò¡À.
M00962	BIT	962.[AoAO¡¤I¢¥o] AoAO ¨¡¢ç¡¤©öAI ¡ío¨¬I 1 A¡þ¡¤¡ÍCA ¢¯¡©¢¬©÷/¢¥YEu ¨ù¨ú¨ù¡© ¨úE¢Ò¡À.
M00963	BIT	963.[AoAO¡¤I¢¥o] AoAO ¨¡¢ç¡¤©öAI ¡ío¨¬I 2 A¡þ¡¤¡ÍCA ¢¯¡©¢¬©÷/¢¥YEu ¨ù¨ú¨ù¡© ¨úE¢Ò¡À.
M00964	BIT	964.[AoAO¡¤I¢¥o] AoAO 1A¡À CC¢¥o ¨ö¨¬AU A¡×A¢® ¨¡¢ç¡¤©öAI ¡Æ¡§Ao ¨úE¥ìE.
M00965	BIT	965.[AoAO¡¤I¢¥o] AoAO ¢¯¢´¢¬¢ç¨¬¡ÌAIAI ¨¡¢ç¡¤©öAI ©öoA¡§ ¨ù¨ú¨ù¡© ¨úE¢Ò¡À.
M00966	BIT	966.[AoAO¡¤I¢¥o] 
M00967	BIT	967.[AoAO¡¤I¢¥o] 
M00968	BIT	968.[AoAO¡¤I¢¥o] 
M00969	BIT	969.[AoAO¡¤I¢¥o] AoAO 2A¡À CC¢¥o XAa ¢¯©ªA¢®¨¬©ö¡¾I ©öI ¢¯I¡¤a.
M0096A	BIT	96A.[AoAO¡¤I¢¥o] AoAO 2A¡À CC¢¥o XAa A¢´¡ío A¡×A¢®¡Æ¢® ¨ú¨¡¢¥O.
M0096B	BIT	96B.[AoAO¡¤I¢¥o] AoAO 2A¡À CC¢¥o XAa ¨ù¡©¨¬¢¬ ¥ìa¢ÒoAI©öo ¢¯¢®¡¤?©ö©¬¡íy. ¢¯¢®¡¤?AU¥ìa E¢çAI©öU¢Ò¡À.
M0096C	BIT	96C.[AoAO¡¤I¢¥o] AoAO 2A¡À CC¢¥o XAa ¨ù¡©¨¬¢¬¢¬©£AI AI¥ì¢¯CIAo ¨úEA¨ö.
M0096D	BIT	96D.[AoAO¡¤I¢¥o] AoAO 2A¡À CC¢¥o XAa ¨ù¡©¨¬¢¬¢¬©£AI +¢¬¢ç©öI¨¡¢ç.
M0096E	BIT	96E.[AoAO¡¤I¢¥o] AoAO 2A¡À CC¢¥o XAa ¨ù¡©¨¬¢¬¢¬©£AI -¢¬¢ç©öI¨¡¢ç.
M0096F	BIT	96F.[AoAO¡¤I¢¥o] AoAO 2A¡À CC¢¥o XAa ¨ù¡©¨¬¢¬ ¢¯ACA.
M00970	BIT	970.[AoAO¡¤I¢¥o] AoAO 2A¡À CC¢¥o A¡þ¡¤¡ÍCA ¢¯¡©¢¬©÷/¢¥YEu ¨ù¨ú¨ù¡© ¨úE¢Ò¡À.
M00971	BIT	971.[AoAO¡¤I¢¥o] AoAO 2A¡À CC¢¥o ¨ö¨¬AU A¡×A¢® ¨¡¢ç¡¤©öAI ¡Æ¡§Ao ¨úE¥ìE.
M00972	BIT	972.[AoAO¡¤I¢¥o] 
M00973	BIT	973.[AoAO¡¤I¢¥o] 
M00974	BIT	974.[AoAO¡¤I¢¥o] 
M00975	BIT	975.[AoAO¡¤I¢¥o] 
M00976	BIT	976.[AoAO¡¤I¢¥o] 
M00977	BIT	977.[AoAO¡¤I¢¥o] 
M00978	BIT	978.[AoAO¡¤I¢¥o] AoAO AUAc CCA¢¯ ©öoA¡§ ¨ù¨ú¨ù¡© ¨úE¢Ò¡À.
M00979	BIT	979.[AoAO¡¤I¢¥o] AoAO AUAc CCA¢¯ YAa ¢¯©ªA¢®¨¬©ö¡¾I ©öI ¢¯I¡¤a.
M0097A	BIT	97A.[AoAO¡¤I¢¥o] AoAO AUAc CCA¢¯ YAa A¢´¡ío A¡×A¢®¡Æ¢® ¨ú¨¡¢¥O.
M0097B	BIT	97B.[AoAO¡¤I¢¥o] AoAO AUAc CCA¢¯ YAa ¨ù¡©¨¬¢¬ ¥ìa¢ÒoAI©öo ¢¯¢®¡¤?©ö©¬¡íy. ¢¯¢®¡¤?AU¥ìa E¢çAI©öU¢Ò¡À.
M0097C	BIT	97C.[AoAO¡¤I¢¥o] AoAO AUAc CCA¢¯ YAa ¨ù¡©¨¬¢¬¢¬©£AI AI¥ì¢¯CIAo ¨úEA¨ö.
M0097D	BIT	97D.[AoAO¡¤I¢¥o] AoAO AUAc CCA¢¯ YAa ¨ù¡©¨¬¢¬¢¬©£AI +¢¬¢ç©öI¨¡¢ç.
M0097E	BIT	97E.[AoAO¡¤I¢¥o] AoAO AUAc CCA¢¯ YAa ¨ù¡©¨¬¢¬¢¬©£AI -¢¬¢ç©öI¨¡¢ç.
M0097F	BIT	97F.[AoAO¡¤I¢¥o] AoAO AUAc CCA¢¯ YAa ¨ù¡©¨¬¢¬ ¢¯ACA.
M00980	BIT	980.[AoAO¡¤I¢¥o] AoAO ¢¯¢´¢¬¢ç¨¬¡ÌAIAI ZAa ¢¯©ªA¢® ¨¬©ö¡¾IA©¬¢®|
M00981	BIT	981.[AoAO¡¤I¢¥o] AoAO 1A¡À CC¢¥o XAa ¢¯©ªA¢® ¨¬©ö¡¾IA©¬¢®|
M00982	BIT	982.[AoAO¡¤I¢¥o] AoAO 2A¡À CC¢¥o XAa ¢¯©ªA¢® ¨¬©ö¡¾IA©¬¢®|
M00983	BIT	983.[AoAO¡¤I¢¥o] AoAO AUAc CCA¢¯ YAa ¢¯©ªA¢® ¨¬©ö¡¾IA©¬¢®|
M00984	BIT	984.[AoAO¡¤I¢¥o] 
M00985	BIT	985.[AoAO¡¤I¢¥o] 
M00986	BIT	986.[AoAO¡¤I¢¥o] 
M00987	BIT	987.[AoAO¡¤I¢¥o] 
M00988	BIT	988.[AoAO¡¤I¢¥o] 
M00989	BIT	989.[AoAO¡¤I¢¥o]
M0098A	BIT	98A.[AoAO¡¤I¢¥o] 
M0098B	BIT	98B.[AoAO¡¤I¢¥o] 
M0098C	BIT	98C.[AoAO¡¤I¢¥o] 
M0098D	BIT	98D.[AoAO¡¤I¢¥o] 
M0098E	BIT	98E.[AoAO¡¤I¢¥o] 
M0098F	BIT	98F.[AoAO¡¤I¢¥o] 
M01020	BIT	1020.[©öeAa¡¤I¢¥o] ¨¬n¡íoA¢´Ao
M01021	BIT	1021.[©öeAa¡¤I¢¥o] ¢¬¨­AI ¢¯¢®¨úi ¡Æ©ª¡¾¨­ ¨úE¢Ò¡À.
M01022	BIT	1022.[©öeAa¡¤I¢¥o] AoAO¨¬I ¨úEAu ¨ù¨ú¨ù¡© ¡Æ¡§Ao¥ìE.
M01023	BIT	1023.[©öeAa¡¤I¢¥o] ©öeAa¨¬I ¨úEAu ¨ù¨ú¨ù¡© ¡Æ¡§Ao¥ìE.
M01024	BIT	1024.[©öeAa¡¤I¢¥o] AoAO¨¬I Au¢¬e ¨úEAu©ö¢ç ¢¯¡©¢¬©÷.
M01025	BIT	1025.[©öeAa¡¤I¢¥o] AoAO¨¬I ¢¯¡¤¢¬e ¨úEAu©ö¢ç ¢¯¡©¢¬©÷.
M01026	BIT	1026.[©öeAa¡¤I¢¥o] ©öeAa¨¬I Au¢¬e ¨úEAu©ö¢ç ¢¯¡©¢¬©÷.
M01027	BIT	1027.[©öeAa¡¤I¢¥o] 
M01028	BIT	1028.[©öeAa¡¤I¢¥o] 
M01029	BIT	1029.[©öeAa¡¤I¢¥o] AoAO ¢¯¢´¢¬¢ç¨¬¡ÌAIAI ZAa ¢¯©ªA¢®¨¬©ö¡¾I ©öI ¢¯I¡¤a.
M0102A	BIT	102A.[©öeAa¡¤I¢¥o] AoAO ¢¯¢´¢¬¢ç¨¬¡ÌAIAI ZAa A¢´¡ío A¡×A¢®¡Æ¢® ¨ú¨¡¢¥O.
M0102B	BIT	102B.[©öeAa¡¤I¢¥o] AoAO ¢¯¢´¢¬¢ç¨¬¡ÌAIAI ZAa ¨ù¡©¨¬¢¬ ¥ìa¢ÒoAI©öo ¢¯¢®¡¤?©ö©¬¡íy. ¢¯¢®¡¤?AU¥ìa E¢çAI©öU¢Ò¡À.
M0102C	BIT	102C.[©öeAa¡¤I¢¥o] AoAO ¢¯¢´¢¬¢ç¨¬¡ÌAIAI ZAoAO ¢¯¢´¢¬¢ç¨¬¡ÌAIAI ZAa ¨ù¡©¨¬¢¬¢¬©£AI AI¥ì¢¯CIAo ¨úEA¨ö.
M0102D	BIT	102D.[©öeAa¡¤I¢¥o] AoAO ¢¯¢´¢¬¢ç¨¬¡ÌAIAI ZAoAO ¢¯¢´¢¬¢ç¨¬¡ÌAIAI ZAa ¨ù¡©¨¬¢¬¢¬©£AI +¢¬¢ç©öI¨¡¢ç.
M0102E	BIT	102E.[©öeAa¡¤I¢¥o] AoAO ¢¯¢´¢¬¢ç¨¬¡ÌAIAI ZAa ¨ù¡©¨¬¢¬¢¬©£AI -¢¬¢ç©öI¨¡¢ç.
M0102F	BIT	102F.[©öeAa¡¤I¢¥o] AoAO ¢¯¢´¢¬¢ç¨¬¡ÌAIAI ZAa ¨ù¡©¨¬¢¬ ¢¯ACA.
M01030	BIT	1030.[©öeAa¡¤I¢¥o] AoAO ¨ù¡©¨¡¡À¨¡¢ç1 ¢¯¡©¢¬©÷/¢¥YEu ¨ù¨ú¨ù¡© ¨úE¢Ò¡À.
M01031	BIT	1031.[©öeAa¡¤I¢¥o] AoAO ¨ù¡©¨¡¡À¨¡¢ç2 ¢¯¡©¢¬©÷/¢¥YEu ¨ù¨ú¨ù¡© ¨úE¢Ò¡À.
M01032	BIT	1032.[©öeAa¡¤I¢¥o] AoAO ¨¡¢ç¡¤©öAI ¨¬¨¢¢¬¢ç1 ¢¯¡©¢¬©÷/¢¥YEu ¨ù¨ú¨ù¡© ¨úE¢Ò¡À.
M01033	BIT	1033.[©öeAa¡¤I¢¥o] AoAO ¨¡¢ç¡¤©öAI ¨¬¨¢¢¬¢ç2 ¢¯¡©¢¬©÷/¢¥YEu ¨ù¨ú¨ù¡© ¨úE¢Ò¡À.
M01034	BIT	1034.[©öeAa¡¤I¢¥o] AoAO ¨¡¢ç¡¤©öAI ©öeAa ¡ío¨öA/CI¡Æ¡© ¨ù¨ú¨ù¡© ¨úE¢Ò¡À.
M01035	BIT	1035.[©öeAa¡¤I¢¥o] AoAO ¨¡¢ç¡¤©öAI ¢¯¢´¢¬¢ç¨¬¡ÌAIAI ¢¯¥ì¢¯¨£ ¡¤©öAIA¡× ¨úEA©ª ¨¬O¡¤¢ç.
M01036	BIT	1036.[©öeAa¡¤I¢¥o] AoAO ¢¯¢´¢¬¢ç¨¬¡ÌAIAI ¡ío¨öA ¡Æ¢®¢¥E ¨ù¨ú¨ù¡© ¨úE¢Ò¡À.
M01037	BIT	1037.[©öeAa¡¤I¢¥o] AoAO ¢¬¢çCA¨¡¢ç ¡ío¨öA ¡Æ¢®¢¥E ¨ù¨ú¨ù¡© ¨úE¢Ò¡À.
M01038	BIT	1038.[©öeAa¡¤I¢¥o] AoAO AU¨ú¡À ¢¯I¡¤a ¨¡¢ç¡¤©öAI ¡Æ¢®¥ì©¡Au.
M01039	BIT	1039.[©öeAa¡¤I¢¥o] AoAO 1A¡À CC¢¥o XAa ¢¯©ªA¢®¨¬©ö¡¾I ©öI ¢¯I¡¤a.
M0103A	BIT	103A.[©öeAa¡¤I¢¥o] AoAO 1A¡À CC¢¥o XAa A¢´¡ío A¡×A¢®¡Æ¢® ¨ú¨¡¢¥O.
M0103B	BIT	103B.[©öeAa¡¤I¢¥o] AoAO 1A¡À CC¢¥o XAa ¨ù¡©¨¬¢¬ ¥ìa¢ÒoAI©öo ¢¯¢®¡¤?©ö©¬¡íy. ¢¯¢®¡¤?AU¥ìa E¢çAI©öU¢Ò¡À.
M0103C	BIT	103C.[©öeAa¡¤I¢¥o] AoAO 1A¡À CC¢¥o XAa ¨ù¡©¨¬¢¬¢¬©£AI AI¥ì¢¯CIAo ¨úEA¨ö.
M0103D	BIT	103D.[©öeAa¡¤I¢¥o] AoAO 1A¡À CC¢¥o XAa ¨ù¡©¨¬¢¬¢¬©£AI +¢¬¢ç©öI¨¡¢ç.
M0103E	BIT	103E.[©öeAa¡¤I¢¥o] AoAO 1A¡À CC¢¥o XAa ¨ù¡©¨¬¢¬¢¬©£AI -¢¬¢ç©öI¨¡¢ç.
M0103F	BIT	103F.[©öeAa¡¤I¢¥o] AoAO 1A¡À CC¢¥o XAa ¨ù¡©¨¬¢¬ ¢¯ACA.
M01040	BIT	1040.[©öeAa¡¤I¢¥o] AoAO 1A¡À CC¢¥o A¡þ¡¤¡ÍCA ¢¯¡©¢¬©÷/¢¥YEu ¨ù¨ú¨ù¡© ¨úE¢Ò¡À.
M01041	BIT	1041.[©öeAa¡¤I¢¥o] AoAO ¨¡¢ç¡¤©öAI ¢¯¡¤ A¡þ¡¤¡ÍCA ¢¯¡©¢¬©÷/¢¥YEu ¨ù¨ú¨ù¡© ¨úE¢Ò¡À.
M01042	BIT	1042.[©öeAa¡¤I¢¥o] AoAO ¨¡¢ç¡¤©öAI ¡ío¨¬I 1 A¡þ¡¤¡ÍCA ¢¯¡©¢¬©÷/¢¥YEu ¨ù¨ú¨ù¡© ¨úE¢Ò¡À.
M01043	BIT	1043.[©öeAa¡¤I¢¥o] AoAO ¨¡¢ç¡¤©öAI ¡ío¨¬I 2 A¡þ¡¤¡ÍCA ¢¯¡©¢¬©÷/¢¥YEu ¨ù¨ú¨ù¡© ¨úE¢Ò¡À.
M01044	BIT	1044.[©öeAa¡¤I¢¥o] AoAO 1A¡À CC¢¥o ¨ö¨¬AU A¡×A¢® ¨¡¢ç¡¤©öAI ¡Æ¡§Ao ¨úE¥ìE.
M01045	BIT	1045.[©öeAa¡¤I¢¥o] AoAO ¢¯¢´¢¬¢ç¨¬¡ÌAIAI ¨¡¢ç¡¤©öAI ©öoA¡§ ¨ù¨ú¨ù¡© ¨úE¢Ò¡À.
M01046	BIT	1046.[©öeAa¡¤I¢¥o] 
M01047	BIT	1047.[©öeAa¡¤I¢¥o] 
M01048	BIT	1048.[©öeAa¡¤I¢¥o] 
M01049	BIT	1049.[©öeAa¡¤I¢¥o] AoAO 2A¡À CC¢¥o XAa ¢¯©ªA¢®¨¬©ö¡¾I ©öI ¢¯I¡¤a.
M0104A	BIT	104A.[©öeAa¡¤I¢¥o] AoAO 2A¡À CC¢¥o XAa A¢´¡ío A¡×A¢®¡Æ¢® ¨ú¨¡¢¥O.
M0104B	BIT	104B.[©öeAa¡¤I¢¥o] AoAO 2A¡À CC¢¥o XAa ¨ù¡©¨¬¢¬ ¥ìa¢ÒoAI©öo ¢¯¢®¡¤?©ö©¬¡íy. ¢¯¢®¡¤?AU¥ìa E¢çAI©öU¢Ò¡À.
M0104C	BIT	104C.[©öeAa¡¤I¢¥o] AoAO 2A¡À CC¢¥o XAa ¨ù¡©¨¬¢¬¢¬©£AI AI¥ì¢¯CIAo ¨úEA¨ö.
M0104D	BIT	104D.[©öeAa¡¤I¢¥o] AoAO 2A¡À CC¢¥o XAa ¨ù¡©¨¬¢¬¢¬©£AI +¢¬¢ç©öI¨¡¢ç.
M0104E	BIT	104E.[©öeAa¡¤I¢¥o] AoAO 2A¡À CC¢¥o XAa ¨ù¡©¨¬¢¬¢¬©£AI -¢¬¢ç©öI¨¡¢ç.
M0104F	BIT	104F.[©öeAa¡¤I¢¥o] AoAO 2A¡À CC¢¥o XAa ¨ù¡©¨¬¢¬ ¢¯ACA.
M01050	BIT	1050.[©öeAa¡¤I¢¥o] AoAO 2A¡À CC¢¥o A¡þ¡¤¡ÍCA ¢¯¡©¢¬©÷/¢¥YEu ¨ù¨ú¨ù¡© ¨úE¢Ò¡À.
M01051	BIT	1051.[©öeAa¡¤I¢¥o] AoAO 2A¡À CC¢¥o ¨ö¨¬AU A¡×A¢® ¨¡¢ç¡¤©öAI ¡Æ¡§Ao ¨úE¥ìE.
M01052	BIT	1052.[©öeAa¡¤I¢¥o] 
M01053	BIT	1053.[©öeAa¡¤I¢¥o] 
M01054	BIT	1054.[©öeAa¡¤I¢¥o] 
M01055	BIT	1055.[©öeAa¡¤I¢¥o] 
M01056	BIT	1056.[©öeAa¡¤I¢¥o] 
M01057	BIT	1057.[©öeAa¡¤I¢¥o] 
M01058	BIT	1058.[©öeAa¡¤I¢¥o] AoAO AUAc CCA¢¯ ©öoA¡§ ¨ù¨ú¨ù¡© ¨úE¢Ò¡À.
M01059	BIT	1059.[©öeAa¡¤I¢¥o] AoAO AUAc CCA¢¯ YAa ¢¯©ªA¢®¨¬©ö¡¾I ©öI ¢¯I¡¤a.
M0105A	BIT	105A.[©öeAa¡¤I¢¥o] AoAO AUAc CCA¢¯ YAa A¢´¡ío A¡×A¢®¡Æ¢® ¨ú¨¡¢¥O.
M0105B	BIT	105B.[©öeAa¡¤I¢¥o] AoAO AUAc CCA¢¯ YAa ¨ù¡©¨¬¢¬ ¥ìa¢ÒoAI©öo ¢¯¢®¡¤?©ö©¬¡íy. ¢¯¢®¡¤?AU¥ìa E¢çAI©öU¢Ò¡À.
M0105C	BIT	105C.[©öeAa¡¤I¢¥o] AoAO AUAc CCA¢¯ YAa ¨ù¡©¨¬¢¬¢¬©£AI AI¥ì¢¯CIAo ¨úEA¨ö.
M0105D	BIT	105D.[©öeAa¡¤I¢¥o] AoAO AUAc CCA¢¯ YAa ¨ù¡©¨¬¢¬¢¬©£AI +¢¬¢ç©öI¨¡¢ç.
M0105E	BIT	105E.[©öeAa¡¤I¢¥o] AoAO AUAc CCA¢¯ YAa ¨ù¡©¨¬¢¬¢¬©£AI -¢¬¢ç©öI¨¡¢ç.
M0105F	BIT	105F.[©öeAa¡¤I¢¥o] AoAO AUAc CCA¢¯ YAa ¨ù¡©¨¬¢¬ ¢¯ACA.
M01060	BIT	1060.[©öeAa¡¤I¢¥o] AoAO ¢¯¢´¢¬¢ç¨¬¡ÌAIAI ZAa ¢¯©ªA¢® ¨¬©ö¡¾IA©¬¢®|
M01061	BIT	1061.[©öeAa¡¤I¢¥o] AoAO 1A¡À CC¢¥o XAa ¢¯©ªA¢® ¨¬©ö¡¾IA©¬¢®|
M01062	BIT	1062.[©öeAa¡¤I¢¥o] AoAO 2A¡À CC¢¥o XAa ¢¯©ªA¢® ¨¬©ö¡¾IA©¬¢®|
M01063	BIT	1063.[©öeAa¡¤I¢¥o] AoAO AUAc CCA¢¯ YAa ¢¯©ªA¢® ¨¬©ö¡¾IA©¬¢®|
M01064	BIT	1064.[©öeAa¡¤I¢¥o] 
M01065	BIT	1065.[©öeAa¡¤I¢¥o] 
M01066	BIT	1066.[©öeAa¡¤I¢¥o] 
M01067	BIT	1067.[©öeAa¡¤I¢¥o] 
M01068	BIT	1068.[©öeAa¡¤I¢¥o] 
M01069	BIT	1069.[©öeAa¡¤I¢¥o]
M0106A	BIT	106A.[©öeAa¡¤I¢¥o] 
M0106B	BIT	106B.[©öeAa¡¤I¢¥o] 
M0106C	BIT	106C.[©öeAa¡¤I¢¥o] 
M0106D	BIT	106D.[©öeAa¡¤I¢¥o] 
M0106E	BIT	106E.[©öeAa¡¤I¢¥o] 
M0106F	BIT	106F.[©öeAa¡¤I¢¥o] 
M1885A	BIT	T)IN-BUFF FPCB ALGN-U/D(work))
M18854	BIT	T)IN-BUFF FPCB ALGN-BWD
M1884A	BIT	T)IN-BUFF ALGN-updn(work)
M18844	BIT	T)IN-BUFF ALGN-BWD
M18847	BIT	T)IN-BUFF ALGN UP/DN
M0850A	BIT	LOT-END KP
M0240C	BIT	IN-BUFF LD REQ(LF)
M0240D	BIT	IN-BUFF LD REQ(RT)
P0015D	BIT	R_4th FPCB SUPPORT UP/DN
M0074F	BIT	R_4th FPCB SUPPORT UP/DN ALARM
M0066F	BIT	L_4th FPCB SUPPORT UP/DN ALARM
M01238	BIT	LEFT ALARM PLS
M01239	BIT	RIGHT ALARM PLS
M1157B	BIT	L_4th ¨úE¢Ò¡À ¨ú¨¡¢¥O
M1407B	BIT	R_4th ¨úE¢Ò¡À ¨ú¨¡¢¥O
M00110	BIT	break hold cylinder p12a
M00111	BIT	p12a hold
M00115	BIT	p15a hold
M00114	BIT	break hold cylinder p15a
T0010	BIT/WORD	delay cyl align 1
T0011	BIT/WORD	delay cyl aligh 1 r
M00060	BIT	cyl align p15d out
P0008F	BIT	R_4th DIE ALIGN BACKWARD
M00061	BIT	cyl align1 -l out
M1217A	BIT	L_P&P Y 2D MOVE_KP
M1467A	BIT	R_P&P Y 2D MOVE_KP
ZR00001	WORD	AUTO STEP IN BUFFER
ZR00002	WORD	AUTO STEP OUT BUFFER
M15000	BIT	AUTO INBUFF STEP#00
M15001	BIT	AUTO INBUFF STEP#01
M15003	BIT	AUTO INBUFF STEP#03
M15004	BIT	AUTO INBUFF STEP#04
M15002	BIT	AUTO INBUFF STEP#02
M15005	BIT	AUTO INBUFF STEP#05
M15006	BIT	AUTO INBUFF STEP#06
M15008	BIT	AUTO INBUFF STEP#08
M15007	BIT	AUTO INBUFF STEP#07
M15009	BIT	AUTO INBUFF STEP#09
M1500A	BIT	AUTO INBUFF STEP#10
M1500B	BIT	AUTO INBUFF STEP#11
M1500C	BIT	AUTO INBUFF STEP#12
M1500D	BIT	AUTO INBUFF STEP#13
M1500E	BIT	AUTO INBUFF STEP#14
M1500F	BIT	AUTO INBUFF STEP#15
M15010	BIT	AUTO INBUFF STEP#16
M15011	BIT	AUTO INBUFF STEP#17
M15012	BIT	AUTO INBUFF STEP#18
M15013	BIT	AUTO INBUFF STEP#19
M15014	BIT	AUTO INBUFF STEP#20
M15015	BIT	AUTO INBUFF STEP#21
M15016	BIT	AUTO INBUFF STEP#22
M15017	BIT	AUTO INBUFF STEP#23
M15018	BIT	AUTO INBUFF STEP#24
M15019	BIT	AUTO INBUFF STEP#25
M1501A	BIT	AUTO INBUFF STEP#26
M1501B	BIT	AUTO INBUFF STEP#27
M1501C	BIT	AUTO INBUFF STEP#28
M1501D	BIT	AUTO INBUFF STEP#29
M1501E	BIT	AUTO INBUFF STEP#30
M1501F	BIT	AUTO INBUFF STEP#31
M15020	BIT	AUTO INBUFF STEP#32
M15021	BIT	AUTO INBUFF STEP#33
M15022	BIT	AUTO INBUFF STEP#34
M15023	BIT	AUTO INBUFF STEP#35
M15024	BIT	AUTO INBUFF STEP#36
M15025	BIT	AUTO INBUFF STEP#37
M15026	BIT	AUTO INBUFF STEP#38
M15027	BIT	AUTO INBUFF STEP#39
M15028	BIT	AUTO INBUFF STEP#40
M15029	BIT	AUTO INBUFF STEP#41
M1502A	BIT	AUTO INBUFF STEP#42
M1502B	BIT	AUTO INBUFF STEP#43
M1502C	BIT	AUTO INBUFF STEP#44
M1502D	BIT	AUTO INBUFF STEP#45
M1502E	BIT	AUTO INBUFF STEP#46
M1502F	BIT	AUTO INBUFF STEP#47
M15030	BIT	AUTO INBUFF STEP#48
M15031	BIT	AUTO INBUFF STEP#49
M15032	BIT	AUTO INBUFF STEP#50
M15033	BIT	AUTO INBUFF STEP#51
M15034	BIT	AUTO INBUFF STEP#52
M15035	BIT	AUTO INBUFF STEP#53
M15036	BIT	AUTO INBUFF STEP#54
M15037	BIT	AUTO INBUFF STEP#55
M15038	BIT	AUTO INBUFF STEP#56
M15039	BIT	AUTO INBUFF STEP#57
M1503A	BIT	AUTO INBUFF STEP#58
M1503B	BIT	AUTO INBUFF STEP#59
M1503C	BIT	AUTO INBUFF STEP#60
M1503D	BIT	AUTO INBUFF STEP#61
M1503E	BIT	AUTO INBUFF STEP#62
M1503F	BIT	AUTO INBUFF STEP#63
M15100	BIT	L_BUFF > L_P&P
M15101	BIT	R_BUFF > R_P&P
T0080	BIT/WORD	ALIGN IN BUFF TIME
M15056	BIT	R_BUFF VACUMN ON [P109]
M15066	BIT	L_BUFF VACUMN ON [P099]
T0081	BIT/WORD	ALIGN IN BUFF TIME
M10298	BIT	T)L_1st_05 Y Pos.3rd
M1029A	BIT	T)L_1st_05 Y Pos.3rd
M12818	BIT	T)R_1st_13 Y Pos.3rd
M1281A	BIT	T)R_1st_13 Y Pos.3rd
T4008	BIT/WORD	L_1st
T4009	BIT/WORD	L_1st
T4010	BIT/WORD	L_1st
T4011	BIT/WORD	L_1st
T4012	BIT/WORD	L_1st
T4013	BIT/WORD	L_1st
T4014	BIT/WORD	L_1st
T4015	BIT/WORD	L_1st
T4016	BIT/WORD	L_1st
T4017	BIT/WORD	L_1st
T4018	BIT/WORD	L_1st
T4019	BIT/WORD	L_1st
T4034	BIT/WORD	L_2nd 
T4035	BIT/WORD	L_2nd 
T4036	BIT/WORD	L_2nd 
T4037	BIT/WORD	L_2nd 
T4038	BIT/WORD	L_2nd 
T4039	BIT/WORD	L_2nd 
T4048	BIT/WORD	L_3rd
T4049	BIT/WORD	L_3rd
T4050	BIT/WORD	L_3rd
T4051	BIT/WORD	L_3rd
T4052	BIT/WORD	L_3rd
T4053	BIT/WORD	L_3rd
T4054	BIT/WORD	L_3rd
T4055	BIT/WORD	L_3rd
T4056	BIT/WORD	L_3rd
T4057	BIT/WORD	L_3rd
T4058	BIT/WORD	L_3rd
T4059	BIT/WORD	L_3rd
T4060	BIT/WORD	L_3rd
T4061	BIT/WORD	L_3rd
T4062	BIT/WORD	L_3rd
T4063	BIT/WORD	L_3rd
T4064	BIT/WORD	L_3rd
T4065	BIT/WORD	L_3rd
T4066	BIT/WORD	L_3rd
T4067	BIT/WORD	L_3rd
T4068	BIT/WORD	L_3rd
T4069	BIT/WORD	L_3rd
T4078	BIT/WORD	L_4th
T4079	BIT/WORD	L_4th
T4080	BIT/WORD	L_4th
T4081	BIT/WORD	L_4th
T4082	BIT/WORD	L_4th
T4083	BIT/WORD	L_4th
T4084	BIT/WORD	L_4th
T4085	BIT/WORD	L_4th
T4086	BIT/WORD	L_4th
T4087	BIT/WORD	L_4th
T4088	BIT/WORD	L_4th
T4089	BIT/WORD	L_4th
T4090	BIT/WORD	L_4th
T4091	BIT/WORD	L_4th
T4092	BIT/WORD	L_4th
T4093	BIT/WORD	L_4th
T4094	BIT/WORD	L_4th
T4095	BIT/WORD	L_4th
T4096	BIT/WORD	L_4th
T4097	BIT/WORD	L_4th
T4098	BIT/WORD	L_4th
T4099	BIT/WORD	L_4th
T4208	BIT/WORD	R_1st
T4209	BIT/WORD	R_1st
T4210	BIT/WORD	R_1st
T4211	BIT/WORD	R_1st
T4212	BIT/WORD	R_1st
T4213	BIT/WORD	R_1st
T4214	BIT/WORD	R_1st
T4215	BIT/WORD	R_1st
T4216	BIT/WORD	R_1st
T4217	BIT/WORD	R_1st
T4218	BIT/WORD	R_1st
T4219	BIT/WORD	R_1st
T4234	BIT/WORD	R_2nd 
T4235	BIT/WORD	R_2nd 
T4236	BIT/WORD	R_2nd 
T4237	BIT/WORD	R_2nd 
T4238	BIT/WORD	R_2nd 
T4239	BIT/WORD	R_2nd 
T4248	BIT/WORD	R_3rd
T4249	BIT/WORD	R_3rd
T4250	BIT/WORD	R_3rd
T4251	BIT/WORD	R_3rd
T4252	BIT/WORD	R_3rd
T4253	BIT/WORD	R_3rd
T4254	BIT/WORD	R_3rd
T4255	BIT/WORD	R_3rd
T4256	BIT/WORD	R_3rd
T4257	BIT/WORD	R_3rd
T4258	BIT/WORD	R_3rd
T4259	BIT/WORD	R_3rd
T4260	BIT/WORD	R_3rd
T4261	BIT/WORD	R_3rd
T4262	BIT/WORD	R_3rd
T4263	BIT/WORD	R_3rd
T4264	BIT/WORD	R_3rd
T4265	BIT/WORD	R_3rd
T4266	BIT/WORD	R_3rd
T4267	BIT/WORD	R_3rd
T4268	BIT/WORD	R_3rd
T4269	BIT/WORD	R_3rd
T4278	BIT/WORD	R_4th
T4279	BIT/WORD	R_4th
T4280	BIT/WORD	R_4th
T4281	BIT/WORD	R_4th
T4282	BIT/WORD	R_4th
T4283	BIT/WORD	R_4th
T4284	BIT/WORD	R_4th
T4285	BIT/WORD	R_4th
T4286	BIT/WORD	R_4th
T4287	BIT/WORD	R_4th
T4288	BIT/WORD	R_4th
T4289	BIT/WORD	R_4th
T4290	BIT/WORD	R_4th
T4291	BIT/WORD	R_4th
T4292	BIT/WORD	R_4th
T4293	BIT/WORD	R_4th
T4294	BIT/WORD	R_4th
T4295	BIT/WORD	R_4th
T4296	BIT/WORD	R_4th
T4297	BIT/WORD	R_4th
T4298	BIT/WORD	R_4th
T4299	BIT/WORD	R_4th
P00066	BIT	R_1st SS MANDREL BW
M03190	BIT	-
M03191	BIT	-
M03192	BIT	-
M03193	BIT	-
M03194	BIT	-
M03195	BIT	-
M03196	BIT	-
M03197	BIT	-
M03198	BIT	-
M03199	BIT	-
M0319A	BIT	-
M0319B	BIT	-
M0319D	BIT	-
M0319E	BIT	-
M0319F	BIT	-
M03200	BIT	-
M03201	BIT	-
M03202	BIT	-
M03203	BIT	-
M03204	BIT	-
M03205	BIT	-
M03206	BIT	-
M03207	BIT	-
M03208	BIT	-
M03209	BIT	-
M0320A	BIT	-
M0320B	BIT	-
M0320D	BIT	-
M0320E	BIT	-
M0320F	BIT	-
M03210	BIT	-
M03211	BIT	-
M03212	BIT	-
M03213	BIT	-
M03214	BIT	-
M03215	BIT	-
M03216	BIT	-
M03217	BIT	-
M03218	BIT	-
M03219	BIT	-
M0321A	BIT	-
M0321B	BIT	-
M0321D	BIT	-
M0321E	BIT	-
M0321F	BIT	-
M03220	BIT	-
M03221	BIT	-
M03222	BIT	-
M03223	BIT	-
M03224	BIT	-
M03225	BIT	-
M03226	BIT	-
M03227	BIT	-
M03228	BIT	-
M03229	BIT	-
M0322A	BIT	-
M0322B	BIT	-
M0322D	BIT	-
M0322E	BIT	-
M0322F	BIT	-
M03230	BIT	-
M03231	BIT	-
M03232	BIT	-
M03233	BIT	-
M03234	BIT	-
M03235	BIT	-
M03236	BIT	-
M03237	BIT	-
M03238	BIT	-
M03239	BIT	-
M0323A	BIT	-
M0323B	BIT	-
M0323D	BIT	-
M0323E	BIT	-
M0323F	BIT	-
M03240	BIT	-
M03241	BIT	-
M03242	BIT	-
M03243	BIT	-
M03244	BIT	-
M03245	BIT	-
M03246	BIT	-
M03247	BIT	-
M03248	BIT	-
M03249	BIT	-
M0324A	BIT	-
M0324B	BIT	-
M0324D	BIT	-
M0324E	BIT	-
M0324F	BIT	-
M03250	BIT	-
M03251	BIT	-
M03252	BIT	-
M03253	BIT	-
M03254	BIT	-
M03255	BIT	-
M03256	BIT	-
M03257	BIT	-
M03258	BIT	-
M03259	BIT	-
M0325A	BIT	-
M0325B	BIT	-
M0325D	BIT	-
M0325E	BIT	-
M0325F	BIT	-
M03260	BIT	-
M03261	BIT	-
M03262	BIT	-
M03263	BIT	-
M03264	BIT	-
M03265	BIT	-
M03266	BIT	-
M03267	BIT	-
M03268	BIT	-
M03269	BIT	-
M0326A	BIT	-
M0326B	BIT	-
M0326D	BIT	-
M0326E	BIT	-
M0326F	BIT	-
M03270	BIT	-
M03271	BIT	-
M03272	BIT	-
M03273	BIT	-
M03274	BIT	-
M03275	BIT	-
M03276	BIT	-
M03277	BIT	-
M03278	BIT	-
M03279	BIT	-
M0327A	BIT	-
M0327B	BIT	-
M0327D	BIT	-
M0327E	BIT	-
M0327F	BIT	-
M03280	BIT	-
M03281	BIT	-
M03282	BIT	-
M03283	BIT	-
M03284	BIT	-
M03285	BIT	-
M03286	BIT	-
M03287	BIT	-
M03288	BIT	-
M03289	BIT	-
M0328A	BIT	-
M0328B	BIT	-
M0328D	BIT	-
M0328E	BIT	-
M0328F	BIT	-
M03290	BIT	-
M03291	BIT	-
M03292	BIT	-
M03293	BIT	-
M03294	BIT	-
M03295	BIT	-
M03296	BIT	-
M03297	BIT	-
M03298	BIT	-
M03299	BIT	-
M0329A	BIT	-
M0329B	BIT	-
M0329D	BIT	-
M0329E	BIT	-
M0329F	BIT	-
M03300	BIT	-
M03301	BIT	-
M03302	BIT	-
M03303	BIT	-
M03304	BIT	-
M03305	BIT	-
M03306	BIT	-
M03307	BIT	-
M03308	BIT	-
M03309	BIT	-
M0330A	BIT	-
M0330B	BIT	-
M0330D	BIT	-
M0330E	BIT	-
M0330F	BIT	-
M03310	BIT	-
M03311	BIT	-
M03312	BIT	-
M03313	BIT	-
M03314	BIT	-
M03315	BIT	-
M03316	BIT	-
M03317	BIT	-
M03318	BIT	-
M03319	BIT	-
M0331A	BIT	-
M0331B	BIT	-
M0331D	BIT	-
M0331E	BIT	-
M0331F	BIT	-
M03320	BIT	-
M03321	BIT	-
M03322	BIT	-
M03323	BIT	-
M03324	BIT	-
M03325	BIT	-
M03326	BIT	-
M03327	BIT	-
M03328	BIT	-
M03329	BIT	-
M0332A	BIT	-
M0332B	BIT	-
M13565	BIT	-
M15050	BIT	IN-BUFF SIDE/TOP INITIAL
M15051	BIT	FPCB SIDE/TOP INITIAL
M15057	BIT	ALIGN SIDE/TOP AUTO [P09A-       P094]
M15058	BIT	ALIGN SIDE/TOP FPCB AUTO [P11D-     P11E]
M15067	BIT	ALIGN SIDE/TOP AUTO [P09A-      P094]
M15068	BIT	ALIGN SIDE/TOP FPCB AUTO [P11D-     P11E]
M16000	BIT	AUTO OUTBUFF STEP#00
M16001	BIT	AUTO OUTBUFF STEP#01
M16002	BIT	AUTO OUTBUFF STEP#02
M16003	BIT	AUTO OUTBUFF STEP#03
M16004	BIT	AUTO OUTBUFF STEP#04
M16005	BIT	AUTO OUTBUFF STEP#05
M16006	BIT	AUTO OUTBUFF STEP#06
M16007	BIT	AUTO OUTBUFF STEP#07
M16008	BIT	AUTO OUTBUFF STEP#08
M16009	BIT	AUTO OUTBUFF STEP#09
M1600A	BIT	AUTO OUTBUFF STEP#10
M1600B	BIT	AUTO OUTBUFF STEP#11
M1600C	BIT	AUTO OUTBUFF STEP#12
M1600D	BIT	AUTO OUTBUFF STEP#13
M1600E	BIT	AUTO OUTBUFF STEP#14
M1600F	BIT	AUTO OUTBUFF STEP#15
M16010	BIT	AUTO OUTBUFF STEP#16
M16011	BIT	AUTO OUTBUFF STEP#17
M16012	BIT	AUTO OUTBUFF STEP#18
M16013	BIT	AUTO OUTBUFF STEP#19
M16014	BIT	AUTO OUTBUFF STEP#20
M16015	BIT	AUTO OUTBUFF STEP#21
M16016	BIT	AUTO OUTBUFF STEP#22
M16017	BIT	AUTO OUTBUFF STEP#23
M16018	BIT	AUTO OUTBUFF STEP#24
M16019	BIT	AUTO OUTBUFF STEP#25
M1601A	BIT	AUTO OUTBUFF STEP#26
M1601B	BIT	AUTO OUTBUFF STEP#27
M1601C	BIT	AUTO OUTBUFF STEP#28
M1601D	BIT	AUTO OUTBUFF STEP#29
M1601E	BIT	AUTO OUTBUFF STEP#30
M1601F	BIT	AUTO OUTBUFF STEP#31
M16020	BIT	AUTO OUTBUFF STEP#32
M16021	BIT	AUTO OUTBUFF STEP#33
M16022	BIT	AUTO OUTBUFF STEP#34
M16023	BIT	AUTO OUTBUFF STEP#35
M16024	BIT	AUTO OUTBUFF STEP#36
M16025	BIT	AUTO OUTBUFF STEP#37
M16026	BIT	AUTO OUTBUFF STEP#38
M16027	BIT	AUTO OUTBUFF STEP#39
M16028	BIT	AUTO OUTBUFF STEP#40
M16029	BIT	AUTO OUTBUFF STEP#41
M1602A	BIT	AUTO OUTBUFF STEP#42
M1602B	BIT	AUTO OUTBUFF STEP#43
M1602C	BIT	AUTO OUTBUFF STEP#44
M1602D	BIT	AUTO OUTBUFF STEP#45
M1602E	BIT	AUTO OUTBUFF STEP#46
M1602F	BIT	AUTO OUTBUFF STEP#47
M16030	BIT	AUTO OUTBUFF STEP#48
M16031	BIT	AUTO OUTBUFF STEP#49
M16032	BIT	AUTO OUTBUFF STEP#50
M16033	BIT	AUTO OUTBUFF STEP#51
M16034	BIT	AUTO OUTBUFF STEP#52
M16035	BIT	AUTO OUTBUFF STEP#53
M16036	BIT	AUTO OUTBUFF STEP#54
M16037	BIT	AUTO OUTBUFF STEP#55
M16038	BIT	AUTO OUTBUFF STEP#56
M16039	BIT	AUTO OUTBUFF STEP#57
M1603A	BIT	AUTO OUTBUFF STEP#58
M1603B	BIT	AUTO OUTBUFF STEP#59
M1603C	BIT	AUTO OUTBUFF STEP#60
M1603D	BIT	AUTO OUTBUFF STEP#61
M1603E	BIT	AUTO OUTBUFF STEP#62
M1603F	BIT	AUTO OUTBUFF STEP#63
M1600	WORD	AUTO OUTBUFF STEP
M1500	WORD	AUTO INBUFF STEP
M16100	BIT	L_BUFF > L_P&P
M16101	BIT	R_BUFF > R_P&P
M16103	BIT	L_BUFF > P&P UNLOAD
M16104	BIT	R_BUFF > P&P UNLOAD
M16051	BIT	-
M16050	BIT	-
T0079	BIT/WORD	ALIGN IN BUFF TIME
M15103	BIT	L_BUFF > P&P      LOAD
M15104	BIT	R_BUFF > P&P     LOAD
M16056	BIT	R_BUFF VACUMN OFF [Pxxx]
M16054	BIT	TRANSFER > L [Pxxx]
M16057	BIT	-
M16058	BIT	-
M16064	BIT	TRANSFER > R [Pxxx]
M16066	BIT	L_BUFF VACUMN OFF [Pxxx]
M16067	BIT	-
M16068	BIT	-
M15080	BIT	IN_BUFF MOV L_P&P >
M15082	BIT	IN_BUFF MOV R_P&P >
M15084	BIT	L_IN BUFF ROTATE LD
M15086	BIT	L_IN BUFF EJECTOR ON
M15088	BIT	R_IN BUFF ROTATE LD
M1508A	BIT	R_IN BUFF EJECTOR ON
M15054	BIT	TRANSFER > L_P&P [P09E]
M15064	BIT	TRANSFER > R_P&P [P09F]
M16080	BIT	OUT_BUFF MOV L_P&P >
M16082	BIT	OUT_BUFF MOV R_P&P >
M16084	BIT	L_OUT BUFF ROTATE ULD
M16086	BIT	L_OUT BUFF EJECTOR ON
M16088	BIT	R_OUT BUFF ROTATE ULD
M1608A	BIT	R_OUT BUFF EJECTOR ON
M30000	BIT	INBUFF<>OUTBUFF
M30001	BIT	INBUFF<>OUTBUFF
D10002	WORD	-
D10001	WORD	-